// TwinCAT 3 PLC project AlarmsHandler
// Title: AlarmsHandler
// Company: Marden Edwards
// Author: Wiktor Pytka
// ProjectVersion: 1.0.0.0
// ProgramVersion: 3.1.4026.19
// libraries:
//   Tc2_MC2, * (Beckhoff Automation GmbH)
//   Tc2_SerialCom, * (Beckhoff Automation GmbH)
//   Tc2_Standard, * (Beckhoff Automation GmbH)
//   Tc2_System, * (Beckhoff Automation GmbH)
//   Tc2_TcpIp, * (Beckhoff Automation GmbH)
//   Tc2_Utilities, * (Beckhoff Automation GmbH)
// project tree:
//   DUTs/METS/ADS Symobol/ E_SYMBOL_AccessState.TcDUT, E_SYMBOL_AdsStates.TcDUT, ST_SYMBOL_AddressInfo.TcDUT (not stored)
//   DUTs/METS/AI Codes And Validation/ E_CodeAI.TcDUT (not stored), E_CodeType.TcDUT, ST_CodeInfo.TcDUT, ST_CodeValidation.TcDUT (not stored), ST_RejectItems.TcDUT, ST_RejectReasonsForCase.TcDUT (not stored), ST_RejectReasonsForOuter.TcDUT (not stored), ST_RejectReasonsForPack.TcDUT (not stored)
//   DUTs/METS/AI Codes And Validation/GS1_Standard/ E_GS1_CodeAIType.TcDUT (not stored), E_GS1_CodeLvl.TcDUT (not stored), ST_GS1_AI_Attributs.TcDUT (not stored), ST_GS1_AI_Definition.TcDUT (not stored), ST_GS1_CodeInfo.TcDUT (not stored), ST_GS1_CodeValidation.TcDUT (not stored), ST_GS1_Decode_AI.TcDUT (not stored)
//   DUTs/METS/Alarms/ E_MessageID.TcDUT, E_MessageType.TcDUT (not stored), ST_AlarmDB.TcDUT (not stored), ST_Alarms.TcDUT (not stored), ST_AlarmSettings.TcDUT, ST_AlarmsTable.TcDUT (not stored), ST_AlarmStatus.TcDUT (not stored), ST_ALARM_Aux.TcDUT (not stored)
//   DUTs/METS/Aliases/ T_CAC_Filename_1.TcDUT (not stored), T_CASE_Barcode_1.TcDUT (not stored), T_Char_1.TcDUT (not stored), T_CHM_Filename_1.TcDUT (not stored), T_CodeBATCH_1.TcDUT (not stored), T_CodeBRAND_1.TcDUT (not stored), T_CodeCRYPTO_1.TcDUT (not stored), T_CodeGTIN_1.TcDUT (not stored), T_CodeMRP_1.TcDUT (not stored), T_CodePIT_1.TcDUT (not stored), T_CodePO_1.TcDUT (not stored), T_CodePRODUCEDATE_1.TcDUT (not stored), T_CodeRSKU_1.TcDUT (not stored), T_CodeURL_1.TcDUT (not stored), T_DB_LongSTRING_1.TcDUT (not stored), T_FileExtension_1.TcDUT (not stored), T_FolderName_1.TcDUT (not stored), T_FolderPath_1.TcDUT (not stored), T_FSS_RejecCode_1.TcDUT (not stored), T_HMI_PACK_Barcode_1.TcDUT (not stored), T_ISO8601Time_1.TcDUT (not stored), T_LongSTRING_1.TcDUT (not stored), T_OAC_Filename_1.TcDUT (not stored), T_OCV_Filename_1.TcDUT (not stored), T_OHM_Filename_1.TcDUT (not stored), T_OUTER_Barcode_1.TcDUT (not stored), T_PACK_Barcode_1.TcDUT (not stored), T_PCM_Filename_1.TcDUT (not stored), T_PositiveDINT_1.TcDUT (not stored), T_PositiveINT_1.TcDUT (not stored), T_ProductDescription_1.TcDUT (not stored), T_RejectCode_1.TcDUT (not stored), T_TimeLog_1.TcDUT (not stored)
//   DUTs/METS/Case/CAC/ E_CAC_State.TcDUT (not stored), ST_CAC_Data.TcDUT (not stored)
//   DUTs/METS/Case/CHM/CHM Data Structure/GenericHierarchy/Case Item Structures/ ST_CaseContent.TcDUT (not stored), ST_CaseIdentity.TcDUT (not stored), ST_CaseItem.TcDUT (not stored)
//   DUTs/METS/Case/CHM/CHM Data Structure/GenericHierarchy/Outer Item Structures/ ST_OuterContent.TcDUT (not stored), ST_OuterIdentity.TcDUT (not stored), ST_OuterItem.TcDUT (not stored)
//   DUTs/METS/Case/CHM/CHM Data Structure/GenericHierarchy/Pack Item Structures/ ST_PackIdentity.TcDUT (not stored), ST_PackItem.TcDUT (not stored)
//   DUTs/METS/Case/CHM/CHM Data Structure/GenericHierarchy/ ST_DefaultIdentity.TcDUT (not stored)
//   DUTs/METS/Case/CHM/CHM Data Structure/ ST_Attributes.TcDUT (not stored), ST_CHM_GenericHierarchy.TcDUT (not stored) (excluded from build), ST_GenericHierarchy.TcDUT (not stored), ST_MessageHeader.TcDUT (not stored)
//   DUTs/METS/Case/CHM/ E_CHM_GeneratorState.TcDUT (not stored), E_CHM_State.TcDUT (not stored), E_CHM_WriteMode.TcDUT (not stored) (excluded from build), ST_CHM_Data.TcDUT (not stored)
//   DUTs/METS/Case/ E_CASE_State.TcDUT (not stored), ST_CasePackerInfo.TcDUT (not stored), ST_CASE_CaseQueue.TcDUT (not stored), ST_CASE_DefferOuter.TcDUT (not stored), ST_CASE_InfeedQueue.TcDUT (not stored), ST_CASE_OperationData.TcDUT (not stored)
//   DUTs/METS/Case/ORCA/ E_ORCA_State.TcDUT (not stored), ST_ORCA_BrandInfo.TcDUT (not stored), ST_ORCA_Data.TcDUT (not stored), ST_ORCA_Outers.TcDUT (not stored), ST_ORCA_ProductInfo.TcDUT (not stored), ST_ORCA_SiteInfo.TcDUT (not stored)
//   DUTs/METS/Device/CX Unit/Device/ E_CX_DeviceState.TcDUT (not stored)
//   DUTs/METS/Device/CX Unit/EtherCAT/ E_CX_EtherCATState.TcDUT (not stored), ST_CX_EtherCATDeviceState.TcDUT (not stored), ST_CX_EtherCATMasterPNetState.TcDUT (not stored), ST_CX_EtherCATMasterState.TcDUT (not stored)
//   DUTs/METS/Device/CX Unit/EtherCAT/Terminal FBs/EBUS/ ST_EBUS_AnalogueDataIn.TcDUT (not stored), ST_EBUS_EtherCATState.TcDUT (not stored)
//   DUTs/METS/Device/CX Unit/EtherCAT/Terminal FBs/KBUS/ E_KBUS_RegisterAccessState.TcDUT (not stored), ST_KBUS_AnalogueDataIn.TcDUT (not stored), ST_KBUS_AnalogueDataOut.TcDUT (not stored), ST_KBUS_KL1501DataIn.TcDUT (not stored), ST_KBUS_KL1501DataOut.TcDUT (not stored), ST_KBUS_KL5001Config.TcDUT (not stored)
//   DUTs/METS/Device/CX Unit/EtherCAT/Terminal FBs/ ST_EtherCATSlaveInfo.TcDUT (not stored), ST_EtherCATStatus.TcDUT (not stored)
//   DUTs/METS/Device/CX Unit/Network/ E_CX_NetworkInfoState.TcDUT (not stored), E_CX_SetAMSNetIDState.TcDUT (not stored), ST_CX_AdapterInfo.TcDUT (not stored), ST_CX_NetworkInfo.TcDUT (not stored)
//   DUTs/METS/Device/CX Unit/NOVRAM/ E_CX_NVDataCtrlState.TcDUT (not stored), E_CX_NVDataOpMode.TcDUT (not stored), E_CX_NVXMLState.TcDUT (not stored), ST_CX_AMSAddress.TcDUT (not stored), ST_CX_EL6080DataIn.TcDUT (not stored), ST_CX_EL6080DataOut.TcDUT (not stored), ST_CX_NVDataBlock.TcDUT (not stored)
//   DUTs/METS/Device/CX Unit/System/ E_CX_HWType.TcDUT (not stored), E_CX_State.TcDUT (not stored)
//   DUTs/METS/Device/Cylinders/ E_CYLINDER_Name.TcDUT (not stored), E_CYLINDER_Position.TcDUT (not stored), ST_CYLINDER_Config.TcDUT (not stored), ST_CYLINDER_Control.TcDUT (not stored), ST_CYLINDER_IN.TcDUT (not stored), ST_CYLINDER_OUT.TcDUT (not stored), ST_CYLINDER_Status.TcDUT (not stored), ST_CYLINDER_TagID.TcDUT (not stored)
//   DUTs/METS/Device/DB/ E_DB_ScanState.TcDUT (not stored), ST_DB_CACDataCtrl.TcDUT (not stored), ST_DB_OACDataCtrl.TcDUT (not stored), ST_DB_OCVDataCtrl.TcDUT (not stored)
//   DUTs/METS/Device/DB/OLD/ ST_DBResult.TcDUT (not stored) (excluded from build), ST_DB_CACCheckCtrl.TcDUT (not stored) (excluded from build), ST_DB_Config.TcDUT (not stored), ST_DB_OACCheckCtrl.TcDUT (not stored) (excluded from build), ST_DB_OCVCheckCtrl.TcDUT (not stored) (excluded from build), ST_DB_PcvCheckCtrl.TcDUT (not stored) (excluded from build), ST_DB_ReportDBCtrl.TcDUT (not stored), ST_DB_ReportResult.TcDUT (not stored)
//   DUTs/METS/Device/Drive/Analog/Config/ ST_AnalogDrive.TcDUT (not stored)
//   DUTs/METS/Device/Drive/Analog/ ST_DriveCtrl.TcDUT (not stored), ST_PhtcCtrl.TcDUT (not stored) (excluded from build)
//   DUTs/METS/Device/Drive/MC2/Axis Control/ E_AXIS_MotionType.TcDUT (not stored), ST_AXIS_Control.TcDUT (not stored), ST_AXIS_IN.TcDUT (not stored), ST_AXIS_OUT.TcDUT (not stored), ST_AXIS_Status.TcDUT (not stored)
//   DUTs/METS/Device/Drive/MC2/Config/ ST_AXIS_Config.TcDUT (not stored)
//   DUTs/METS/Device/Drive/MC2/EtherCAT/AX5000 FBs/ ST_AX5000_TouchProbe.TcDUT (not stored)
//   DUTs/METS/Device/Drive/MC2/EtherCAT/Encoder FBs/ ST_DeviceAddress.TcDUT (not stored)
//   DUTs/METS/Device/Drive/MC2/ E_MC_Name.TcDUT (not stored)
//   DUTs/METS/Device/Drive/MC2/NC Axis/Cam/ E_CAM_Update.TcDUT (not stored)
//   DUTs/METS/Device/Drive/MC2/NC Axis/ E_AXIS_CtrlState.TcDUT (not stored), E_TORQUE_Scaling.TcDUT (not stored), ST_AxisCtrlRamps.TcDUT (not stored), ST_DriveStatus.TcDUT (not stored), ST_LatchPosBuffer.TcDUT (not stored), ST_NC_EncDataIn.TcDUT (not stored), ST_NC_EncDataOut.TcDUT (not stored)
//   DUTs/METS/Device/Drive/MC2/TempAxis/ ST_AxisHomeStruct.TcDUT (not stored) (excluded from build), ST_AxisMotionStruct.TcDUT (not stored) (excluded from build)
//   DUTs/METS/Device/Drive/Profinet/Config/ ST_ProfinetDrive.TcDUT (not stored), ST_ProfinetMasterConfig.TcDUT (not stored)
//   DUTs/METS/Device/Drive/Profinet/ E_DRIVE_Name.TcDUT (not stored), ST_PNetMasterStatus.TcDUT (not stored)
//   DUTs/METS/Device/Drive/Profinet/Parameters/ ST_DataPntAdr.TcDUT (not stored), ST_KeyPadDisplay.TcDUT (not stored), ST_Parameter.TcDUT (not stored), ST_ParameterControl.TcDUT (not stored), ST_Parameters.TcDUT (not stored), ST_Value.TcDUT (not stored)
//   DUTs/METS/Device/Drive/Profinet/_G120/Drives/ E_DRIVE_DataType.TcDUT (not stored), ST_DRIVE_INPUT.TcDUT (not stored), ST_DRIVE_OUTPUT.TcDUT (not stored), ST_DRIVE_STATUS.TcDUT (not stored), ST_G120_ExtendedIn.TcDUT (not stored), ST_G120_ExtendedOut.TcDUT (not stored), ST_G120_IN.TcDUT (not stored), ST_G120_OUT.TcDUT (not stored), ST_G120_Status.TcDUT (not stored)
//   DUTs/METS/Device/Drive/Profinet/_G120/ ST_G120_Control.TcDUT (not stored)
//   DUTs/METS/Device/Encoders/CAMS/ ST_AFS60_Cam.TcDUT (not stored), ST_AFS60_CamHMi.TcDUT (not stored), ST_AFS60_Config.TcDUT (not stored), ST_AFS60_Status.TcDUT (not stored)
//   DUTs/METS/Device/Encoders/ E_ENOCDER_Name.TcDUT (not stored), ST_ENCODER_IN.TcDUT (not stored), ST_ENCODER_OUT.TcDUT (not stored), ST_ENCODER_Status.TcDUT (not stored)
//   DUTs/METS/Device/IO2 Controls/ E_IO2_InputSource.TcDUT (not stored), E_IO2_Type.TcDUT (not stored), ST_IO2_Diagnostic.TcDUT (not stored), ST_IO2_InputPLC.TcDUT (not stored), ST_IO2_OutputPLC.TcDUT (not stored)
//   DUTs/METS/Device/IO2 Controls/Input Ctrl/ ST_IO2_DoubleInputCtrl.TcDUT (not stored), ST_IO2_DoubleInputLockedCtrl.TcDUT (not stored), ST_IO2_SingleInputCtrl.TcDUT (not stored), ST_IO2_SingleInputLockedCtrl.TcDUT (not stored)
//   DUTs/METS/Device/IO2 Controls/Outpout Ctrl/ ST_IO2_OutputCtrl.TcDUT (not stored)
//   DUTs/METS/Device/Printers/ E_PRINTER_Name.TcDUT (not stored), E_PRINTER_State.TcDUT (not stored), ST_PRINTER_Config.TcDUT (not stored), ST_PRINTER_IN.TcDUT (not stored), ST_PRINTER_OUT.TcDUT (not stored), ST_PRINTER_Status.TcDUT (not stored)
//   DUTs/METS/Device/Scanner/ E_ClientSteps.TcDUT (not stored), E_DataExchaSteps.TcDUT (not stored), E_SCANNER_CodeType.TcDUT (not stored), E_SCANNER_DeviceType.TcDUT (not stored), E_SCANNER_Name.TcDUT (not stored), E_SCANNER_State.TcDUT (not stored), E_SCANNER_Vendor.TcDUT (not stored), ST_SCANNER.TcDUT (not stored), ST_SCANNER_ApplicationIdentifier.TcDUT (not stored), ST_SCANNER_CameraMap.TcDUT (not stored), ST_SCANNER_CodeData.TcDUT (not stored), ST_SCANNER_Config.TcDUT (not stored), ST_SCANNER_Evaluation.TcDUT (not stored), ST_SCANNER_ImageData.TcDUT (not stored), ST_SCANNER_ManualCtrl.TcDUT (not stored), ST_SCANNER_OpState.TcDUT (not stored), ST_SCANNER_Options.TcDUT (not stored), ST_SCANNER_Performance.TcDUT (not stored), ST_SCANNER_Statistics.TcDUT (not stored), ST_SCANNER_TriggerID.TcDUT (not stored)
//   DUTs/METS/Device/Scanner/Hand Scanner/ E_ConnectSteps.TcDUT (not stored), E_DataSequence.TcDUT (not stored), E_SCANNER_Baudrate.TcDUT (not stored), ST_SCANNER_HoneywellConfig.TcDUT (not stored), ST_SCANNER_HoneywellCtrl.TcDUT (not stored), ST_SCANNER_HoneywellStatus.TcDUT (not stored), ST_SCANNER_HostAck.TcDUT (not stored), ST_SCANNER_USBConfig.TcDUT (not stored)
//   DUTs/METS/Device/Scanner/NewModel/ ST_SCANNER_Configuration.TcDUT, ST_SCANNER_Ctrl.TcDUT (not stored), ST_SCANNER_CtrlMapping.TcDUT (not stored), ST_SCANNER_CtrlOptions.TcDUT (not stored) (excluded from build), ST_SCANNER_IN.TcDUT (not stored), ST_SCANNER_ManualStatus.TcDUT (not stored), ST_SCANNER_OUT.TcDUT (not stored), ST_SCANNER_Status.TcDUT (not stored)
//   DUTs/METS/Files/ E_FILE_CtrlState.TcDUT (not stored), E_FILE_DeleteOldFilesState.TcDUT (not stored), E_FILE_State.TcDUT (not stored), ST_FILE_WriteFileStatistic.TcDUT (not stored)
//   DUTs/METS/HMI/Device Manual Control/ ST_HMI_AxisCtrl.TcDUT (not stored), ST_HMI_CylinderCtrl.TcDUT (not stored), ST_HMI_G120Ctrl.TcDUT (not stored), ST_HMI_PrinterCtrl.TcDUT (not stored)
//   DUTs/METS/HMI/Device Status/ E_HMI_DriveStatus.TcDUT, ST_HMI_AxisStatus.TcDUT (not stored), ST_HMI_CylinderStatus.TcDUT (not stored), ST_HMI_G120Status.TcDUT (not stored), ST_HMI_HoneywellStatus.TcDUT (not stored), ST_HMI_PrinterStatus.TcDUT (not stored)
//   DUTs/METS/HMI/HMIQueue/ ST_HMI_CAC_Data.TcDUT (not stored), ST_HMI_CaseRejectCode.TcDUT (not stored), ST_HMI_CaseVerifiedCode.TcDUT (not stored), ST_HMI_CASE_CaseQueue.TcDUT (not stored), ST_HMI_InfeedQueue.TcDUT (not stored), ST_HMI_OAC_Data.TcDUT (not stored), ST_HMI_OCV_Data.TcDUT (not stored), ST_HMI_OuterStatus.TcDUT (not stored), ST_HMI_PACK_BufferStatus.TcDUT (not stored), ST_HMI_PLAS_Queue.TcDUT (not stored)
//   DUTs/METS/HMI/ ST_HMI_BarGraph.TcDUT (not stored), ST_HMI_Buttons.TcDUT (not stored), ST_HMI_CSVStoreTable.TcDUT (not stored), ST_HMI_StationStatus.TcDUT (not stored), ST_HMI_Visualisation.TcDUT (not stored)
//   DUTs/METS/KPI/ ST_KPI_CasePackerSignals.TcDUT (not stored), ST_KPI_CodePos.TcDUT (not stored), ST_KPI_InspectionEfficency.TcDUT (not stored), ST_KPI_ItemsProduced.TcDUT (not stored), ST_KPI_OCVFile.TcDUT (not stored), ST_KPI_OutersProcessing.TcDUT (not stored), ST_KPI_OutersProduced.TcDUT (not stored)
//   DUTs/METS/LogData/ E_LOG_Handler.TcDUT (not stored), ST_LOG_Alarms.TcDUT (not stored), ST_LOG_EventData.TcDUT (not stored), ST_LOG_FileWriteError.TcDUT (not stored), ST_LOG_MachineState.TcDUT (not stored), ST_LOG_RejectReasons.TcDUT (not stored), ST_LOG_WriteImageData.TcDUT (not stored)
//   DUTs/METS/NV Data/ ST_NOVRAM_METS_Cameras.TcDUT (not stored), ST_NOVRAM_METS_CaseInspactionLog.TcDUT (not stored), ST_NOVRAM_METS_DualInputs.TcDUT (not stored), ST_NOVRAM_METS_EventCounters.TcDUT (not stored), ST_NOVRAM_METS_Inspection.TcDUT (not stored)
//   DUTs/METS/Outers/ E_OUTER_AgrregationState.TcDUT (not stored), E_OUTER_State.TcDUT (not stored), ST_OUTER_Status.TcDUT (not stored)
//   DUTs/METS/Outers/OAC/ E_OAC_State.TcDUT (not stored), ST_OAC_Data.TcDUT (not stored)
//   DUTs/METS/Outers/SFLX/ E_SIDEFLEX_UnitType.TcDUT (not stored), ST_SIDEFLEX_Offset.TcDUT (not stored), ST_SIDEFLEX_ProcessData.TcDUT (not stored)
//   DUTs/METS/Packs/ E_OCV_CheckMode.TcDUT (not stored), E_OCV_State.TcDUT (not stored), E_PACK_FilledInStatus.TcDUT (not stored), E_PACK_ReadStep.TcDUT (not stored), E_PACK_State.TcDUT (not stored), ST_PACK_CodeBuffer.TcDUT (not stored), ST_PACK_CodeStatus.TcDUT (not stored), ST_PACK_ConfirmationQueue.TcDUT (not stored), ST_PACK_Data.TcDUT (not stored), ST_PACK_DuplicatesCheck.TcDUT (not stored), ST_PACK_InfeedQueue.TcDUT (not stored), ST_PACK_InTransferQueue.TcDUT (not stored), ST_PACK_LastFilledCodes.TcDUT (not stored), ST_PACK_TriggerOffset.TcDUT (not stored)
//   DUTs/METS/Packs/_Lab/ ST_LAB_OuterData.TcDUT (not stored), ST_LAB_PackData.TcDUT (not stored)
//   DUTs/METS/PCM/ E_PCM_State.TcDUT (not stored), ST_PCM_Data.TcDUT (not stored), ST_PCM_Status.TcDUT (not stored)
//   DUTs/METS/PCM/PCM_Hierarchy/ProductInformation/Product/ ST_HierarchyData.TcDUT (not stored), ST_HierarchyDataList.TcDUT (not stored)
//   DUTs/METS/PCM/PCM_Hierarchy/ProductInformation/Settings/ ST_ToleranceThresholdCS.TcDUT (not stored), ST_ToleranceThresholdOUT.TcDUT (not stored), ST_ToleranceThresholdPK.TcDUT (not stored)
//   DUTs/METS/PCM/PCM_Hierarchy/ProductInformation/ ST_PCMProduct.TcDUT (not stored), ST_PCMSettings.TcDUT (not stored)
//   DUTs/METS/PCM/PCM_Hierarchy/ ST_PCMMessageHeader.TcDUT (not stored), ST_ProductInformation.TcDUT (not stored)
//   DUTs/METS/String Processing/ E_STRING_ExtrMode.TcDUT (not stored)
//   DUTs/METS/System/ E_SYSTEM_CTState.TcDUT (not stored), E_SYSTEM_HandScannerBaudrate.TcDUT (not stored), E_SYSTEM_ItemType.TcDUT (not stored), E_SYSTEM_MachineState.TcDUT (not stored), E_SYSTEM_MaintainFolders.TcDUT (not stored), E_SYSTEM_OSType.TcDUT (not stored), ST_SYSTEM_Config.TcDUT, ST_SYSTEM_DateTime.TcDUT (not stored), ST_SYSTEM_DeviceState.TcDUT (not stored), ST_SYSTEM_Door.TcDUT (not stored), ST_SYSTEM_MachineID.TcDUT (not stored), ST_SYSTEM_MachineMode.TcDUT (not stored), ST_SYSTEM_MachineState.TcDUT (not stored), ST_SYSTEM_ProductionLine.TcDUT (not stored), ST_SYSTEM_SafetyStatus.TcDUT (not stored), ST_SYSTEM_SoftwareVersion.TcDUT (not stored)
//   DUTs/METS/System/Status/ ST_SYSTEM_ArchiveDBStatus.TcDUT (not stored), ST_SYSTEM_BridgeStatus.TcDUT (not stored), ST_SYSTEM_LoggerStatus.TcDUT (not stored), ST_SYSTEM_MachineStatus.TcDUT (not stored), ST_SYSTEM_ReportingDBStatus.TcDUT (not stored)
//   DUTs/METS/System/System Modes/ E_SYSTEM_AutomationMode.TcDUT (not stored), E_SYSTEM_OuterAggregationMode.TcDUT (not stored), E_SYSTEM_PackAggregationMode.TcDUT (not stored)
//   DUTs/METS/TCPIP Address/ E_TCPIP_State.TcDUT, ST_TCPIP_AddressPort.TcDUT (not stored)
//   DUTs/METS/XML Processing/ E_XML_CtrlState.TcDUT (not stored), E_XML_GeneratorState.TcDUT (not stored), E_XML_WritingMode.TcDUT (not stored)
//   DUTs/METS/_StationOperational/C715 Tempalate Example/ E_04_ElevatorState_C715.TcDUT (not stored), E_Axis_C715.TcDUT (not stored), E_Cylinder_C715.TcDUT (not stored), ST_04_ElevatorSeq_C715.TcDUT (not stored), ST_BundleTrackingRegister_C715.TcDUT (not stored), ST_CommonStationConfig_C715.TcDUT (not stored)
//   DUTs/METS/_StationOperational/ E_00_StationStateTemplate.TcDUT (not stored), ST_00_StationStructTemplate.TcDUT (not stored)
//   DUTs/METS/_StationOperational/Manual Machine/ E_OuterPrintStationState.TcDUT (not stored), ST_OuterPrintStationStruct.TcDUT (not stored)
//   DUTs/METS/_StationOperational/SeqCtrl/ ST_STATION_Requests.TcDUT (not stored), ST_STATION_Status.TcDUT (not stored)
//   GVLs/Global Variables/Aliases/ T_CAC_Filename.TcDUT, T_CASE_Barcode.TcDUT, T_Char.TcDUT, T_CHM_Filename.TcDUT, T_CodeBATCH.TcDUT, T_CodeBRAND.TcDUT, T_CodeCRYPTO.TcDUT, T_CodeGTIN.TcDUT, T_CodeMRP.TcDUT, T_CodePIT.TcDUT, T_CodePO.TcDUT, T_CodePRODUCEDATE.TcDUT, T_CodeRSKU.TcDUT, T_CodeURL.TcDUT, T_DB_LongSTRING.TcDUT, T_FileExtension.TcDUT, T_FolderName.TcDUT, T_FolderPath.TcDUT, T_FSS_RejecCode.TcDUT, T_HMI_PACK_Barcode.TcDUT, T_ISO8601Time.TcDUT, T_LongSTRING.TcDUT, T_OAC_Filename.TcDUT, T_OCV_Filename.TcDUT, T_OHM_Filename.TcDUT, T_OUTER_Barcode.TcDUT, T_PACK_Barcode.TcDUT, T_PCM_Filename.TcDUT, T_PositiveDINT.TcDUT, T_PositiveINT.TcDUT, T_ProductDescription.TcDUT, T_RejectCode.TcDUT, T_TimeLog.TcDUT
//   GVLs/Global Variables/ gConstants.TcGVL (not stored), gHMI.TcGVL (not stored), gIOFiltered.TcGVL (not stored), gMessage.TcGVL, gNovRAM.TcGVL (not stored), gPersistent.TcGVL (not stored)
//   GVLs/Global Variables/InputsOutputsDT/ gCamDevice.TcGVL (not stored), IOVarDT_H.TcGVL (not stored), IOVarDT_S.TcGVL (not stored), _Labs.TcGVL (not stored)
//   GVLs/Global Variables/InputsOutputs_CML/ IOVariablesCX_CML.TcGVL (excluded from build), IOVariablesEUCA_CML.TcGVL (excluded from build), IOVariablesPACAN_CML.TcGVL (excluded from build), IOVariablesPAOL_CML.TcGVL (excluded from build), IOVariablesPLAS_CML.TcGVL (excluded from build)
//   GVLs/Global Variables/InputsOutputs_OC/ IOVariablesCX_OC.TcGVL (excluded from build), IOVariablesEUCA_OC.TcGVL (excluded from build), IOVariablesPAOL_OC.TcGVL (excluded from build), IOVariablesPLAS_OC.TcGVL (excluded from build)
//   GVLs/Global Variables/InputsOutputs_SFLX/ IOVariablesCX_SFLX.TcGVL (excluded from build), IOVariablesEUCA_SFLX.TcGVL (excluded from build), IOVariablesPAOL_SFLX.TcGVL (excluded from build), IOVariablesPLAS_SFLX.TcGVL (excluded from build)
//   GVLs/Global Variables/METS/ gDevice.TcGVL (not stored), gProcess.TcGVL (not stored)
//   GVLs/Global Variables/_VERSION/ _VERSION_CONTROL.TcGVL
//   POUs/Alarm/ FB_ALARM_GroupManagment.TcPOU (not stored), FB_ALARM_Handler.TcPOU (not stored), FB_ALARM_LogTable.TcPOU (not stored), F_ALARM_SetDefinition.TcPOU
//   POUs/Utilities/Concat Function/ F_CONCAT3.TcPOU (not stored), F_CONCAT4.TcPOU (not stored), F_CONCAT5.TcPOU (not stored), F_CONCAT6.TcPOU (not stored), F_CONCAT7.TcPOU (not stored), F_CONCAT8.TcPOU (not stored), F_CONCAT9.TcPOU (not stored)
//   Version/ Global_Version.TcGVL
// real-time tasks:
//   TASK TcUnit_Task: cycle T#10ms, priority 10, ADS port 350

// ---- DUTs/METS/ADS Symobol/E_SYMBOL_AccessState.TcDUT
{attribute 'qualified_only'}
TYPE E_SYMBOL_AccessState :
(
	E_SYMBOL_IDLE,
	E_SYMBOL_GETSYMBOLINFO,
	E_SYMBOL_READDATA,
	E_SYMBOL_WRITEDATA,
	E_SYMBOL_DONE
);
END_TYPE

// ---- DUTs/METS/ADS Symobol/E_SYMBOL_AdsStates.TcDUT
{attribute 'qualified_only'}
TYPE E_SYMBOL_AdsStates :
(
	ADSSTATES_INVALID :=0,
	ADSSTATES_IDLE :=1,
	ADSSTATES_RESET :=2,
	ADSSTATES_INIT :=3,
	ADSSTATES_START :=4,
	ADSSTATES_RUN :=5,
	ADSSTATES_STOP :=6,
	ADSSTATES_SAVECFG :=7,
	ADSSTATES_LOADCFG :=8,
	ADSSTATES_POWERFAILURE :=9,
	ADSSTATES_POWERGOOD :=10,
	ADSSTATES_ERROR :=11
);
END_TYPE

// ---- DUTs/METS/AI Codes And Validation/E_CodeType.TcDUT
{attribute 'qualified_only'}
TYPE E_CodeType :
(
	E_NONE,
	E_PACK,
	E_INTERIM,
	E_OUTER,
	E_CASE
);
END_TYPE

// ---- DUTs/METS/AI Codes And Validation/ST_CodeInfo.TcDUT
TYPE ST_CodeInfo :
STRUCT
	eCodeType					:	E_CodeType;

	nMinLength					: 	INT;
	nEntireLength				:	INT;
	bValidateEntireLength		: 	BOOL;
	nNumberOfAIs				:	INT;

	stGTIN 						:	ST_CodeValidation	:=		(sFieldName :='GTIN',				bNameEditable := FALSE, 	nGS1_AI := 1);
	stBatchID 					:	ST_CodeValidation	:=		(sFieldName :='BatchID', 			bNameEditable := FALSE, 	nGS1_AI := 10);
	stSerialCode 				:	ST_CodeValidation	:=		(sFieldName :='SerialCode', 		bNameEditable := FALSE, 	nGS1_AI := 21);
	stProductionOrder 			:	ST_CodeValidation	:=		(sFieldName :='ProductionOrder', 	bNameEditable := FALSE, 	nGS1_AI := 91);
	stCryptoCode				:	ST_CodeValidation	:=		(sFieldName :='CryptoCode', 		bNameEditable := FALSE, 	nGS1_AI := 93);
	stRSKU						:	ST_CodeValidation	:=		(sFieldName :='RSKU', 				bNameEditable := FALSE, 	nGS1_AI := 240);
	stMRP		 				:	ST_CodeValidation	:=		(sFieldName :='MRP', 				bNameEditable := FALSE, 	nGS1_AI := 8005);
	stBrandSpecification		:	ST_CodeValidation	:=		(sFieldName :='BrandSpec',			bNameEditable := FALSE, 	nGS1_AI := 92);
	stProduceDate				:	ST_CodeValidation	:=		(sFieldName :='ProduceDate',		bNameEditable := TRUE, 		nGS1_AI := 94);
	stUserField					:	ST_CodeValidation	:=		(sFieldName :='',					bNameEditable := TRUE, 		nGS1_AI := 95);

END_STRUCT
END_TYPE

// ---- DUTs/METS/AI Codes And Validation/ST_RejectItems.TcDUT
TYPE ST_RejectItems :
STRUCT
	nRejectID			: UINT;
	sMetsDisplayCode	: T_RejectCode; (*this is what is displayed on our HMI - nn is replaced by the number of failures/successes*)
	sMetsSearchCode	: STRING(50); (*this is what to search for when changing the reject reason for FSS*)
	sFssSendCode		: T_FSS_RejecCode; (*this is what to send to FSS*)
END_STRUCT
END_TYPE

// ---- DUTs/METS/Alarms/E_MessageID.TcDUT
{attribute 'qualified_only'}
{attribute 'to_string'}
TYPE E_MessageID :
(
	MSG_000 := 0,
	MSG_001,
	MSG_002,
	MSG_003,
	MSG_004,
	MSG_005,
	MSG_006,
	MSG_007,
	MSG_008,
	MSG_009,
	MSG_010,
	MSG_011,
	MSG_012,
	MSG_013,
	MSG_014,
	MSG_015,
	MSG_016,
	MSG_017,
	MSG_018,
	MSG_019,
	MSG_020,
	MSG_021,
	MSG_022,
	MSG_023,
	MSG_024,
	MSG_025,
	MSG_026,
	MSG_027,
	MSG_028,
	MSG_029,
	MSG_030,
	MSG_031,
	MSG_032,
	MSG_033,
	MSG_034,
	MSG_035,
	MSG_036,
	MSG_037,
	MSG_038,
	MSG_039,
	MSG_040,
	MSG_041,
	MSG_042,
	MSG_043,
	MSG_044,
	MSG_045,
	MSG_046,
	MSG_047,
	MSG_048,
	MSG_049,
	MSG_050,
	MSG_051,
	MSG_052,
	MSG_053,
	MSG_054,
	MSG_055,
	MSG_056,
	MSG_057,
	MSG_058,
	MSG_059,
	MSG_060,
	MSG_061,
	MSG_062,
	MSG_063,
	MSG_064,
	MSG_065,
	MSG_066,
	MSG_067,
	MSG_068,
	MSG_069,
	MSG_070,
	MSG_071,
	MSG_072,
	MSG_073,
	MSG_074,
	MSG_075,
	MSG_076,
	MSG_077,
	MSG_078,
	MSG_079,
	MSG_080,
	MSG_081,
	MSG_082,
	MSG_083,
	MSG_084,
	MSG_085,
	MSG_086,
	MSG_087,
	MSG_088,
	MSG_089,
	MSG_090,
	MSG_091,
	MSG_092,
	MSG_093,
	MSG_094,
	MSG_095,
	MSG_096,
	MSG_097,
	MSG_098,
	MSG_099,
	MSG_100,
	MSG_101,
	MSG_102,
	MSG_103,
	MSG_104,
	MSG_105,
	MSG_106,
	MSG_107,
	MSG_108,
	MSG_109,
	MSG_110,
	MSG_111,
	MSG_112,
	MSG_113,
	MSG_114,
	MSG_115,
	MSG_116,
	MSG_117,
	MSG_118,
	MSG_119,
	MSG_120,
	MSG_121,
	MSG_122,
	MSG_123,
	MSG_124,
	MSG_125,
	MSG_126,
	MSG_127,
	MSG_128,
	MSG_129,
	MSG_130,
	MSG_131,
	MSG_132,
	MSG_133,
	MSG_134,
	MSG_135,
	MSG_136,
	MSG_137,
	MSG_138,
	MSG_139,
	MSG_140,
	MSG_141,
	MSG_142,
	MSG_143,
	MSG_144,
	MSG_145,
	MSG_146,
	MSG_147,
	MSG_148,
	MSG_149,
	MSG_150,
	MSG_151,
	MSG_152,
	MSG_153,
	MSG_154,
	MSG_155,
	MSG_156,
	MSG_157,
	MSG_158,
	MSG_159,
	MSG_160,
	MSG_161,
	MSG_162,
	MSG_163,
	MSG_164,
	MSG_165,
	MSG_166,
	MSG_167,
	MSG_168,
	MSG_169,
	MSG_170,
	MSG_171,
	MSG_172,
	MSG_173,
	MSG_174,
	MSG_175,
	MSG_176,
	MSG_177,
	MSG_178,
	MSG_179,
	MSG_180,
	MSG_181,
	MSG_182,
	MSG_183,
	MSG_184,
	MSG_185,
	MSG_186,
	MSG_187,
	MSG_188,
	MSG_189,
	MSG_190,
	MSG_191,
	MSG_192,
	MSG_193,
	MSG_194,
	MSG_195,
	MSG_196,
	MSG_197,
	MSG_198,
	MSG_199,
	MSG_200,
	MSG_201,
	MSG_202,
	MSG_203,
	MSG_204,
	MSG_205,
	MSG_206,
	MSG_207,
	MSG_208,
	MSG_209,
	MSG_210,
	MSG_211,
	MSG_212,
	MSG_213,
	MSG_214,
	MSG_215,
	MSG_216,
	MSG_217,
	MSG_218,
	MSG_219,
	MSG_220,
	MSG_221,
	MSG_222,
	MSG_223,
	MSG_224,
	MSG_225,
	MSG_226,
	MSG_227,
	MSG_228,
	MSG_229,
	MSG_230,
	MSG_231,
	MSG_232,
	MSG_233,
	MSG_234,
	MSG_235,
	MSG_236,
	MSG_237,
	MSG_238,
	MSG_239,
	MSG_240,
	MSG_241,
	MSG_242,
	MSG_243,
	MSG_244,
	MSG_245,
	MSG_246,
	MSG_247,
	MSG_248,
	MSG_249,
	MSG_250,
	MSG_251,
	MSG_252,
	MSG_253,
	MSG_254,
	MSG_255
	
);
END_TYPE

// ---- DUTs/METS/Alarms/ST_AlarmSettings.TcDUT
TYPE ST_AlarmSettings :
STRUCT
	aTextMessageTable		: ARRAY [0..31] OF STRING(200);
	aAlarmTriggerTable		: ARRAY [0..31] OF BOOL;

	aAlarmTimoutTable		: ARRAY [0..31] OF TIME;
	aBlockEnableTable		: ARRAY [0..31] OF BOOL :=[ 32 (FALSE)];
	aInhibitResetTable		: ARRAY [0..31] OF BOOL;
	aAutoResetTable			: ARRAY[0..31] OF BOOL;
	//aInternalResetTable		: ARRAY [0..31] OF BOOL;

	aCategoryNoTable		: ARRAY[0..31] OF INT;
	aMessageTypeStatusTable	: ARRAY[0..31] OF WORD;
END_STRUCT
END_TYPE

// ---- DUTs/METS/Device/Scanner/NewModel/ST_SCANNER_Configuration.TcDUT
TYPE ST_SCANNER_Configuration :     //ST_SCANNER_Config
STRUCT
	sDeviceName				: STRING(30) := 'Camera';
	bDisableCameraUse		: BOOL;
	aCameraWarningLevel		: INT := 90;
	stCameraIP				: ST_TCPIP_AddressPort;
	tTimeOut				: TIME := T#3S;
	eCameraVendor			: E_SCANNER_Vendor;
	sFC1ReplacmentChar		: T_Char;
	bDontParseAsGS1			: BOOL;

	eScannerType			: E_SCANNER_DeviceType;
	eExpectedType			: E_SCANNER_CodeType;
	bUseExternalLight		: BOOL;
	nLightingIntensity		: INT;
	nDisplayDelayConfig		: BOOL;

	nImageBuffer			: INT := 1;
	nExpectedResp			: INT := 1;
END_STRUCT
END_TYPE

// ---- DUTs/METS/HMI/Device Status/E_HMI_DriveStatus.TcDUT
{attribute 'qualified_only'}
TYPE E_HMI_DriveStatus :
(
	UNKNOWN := 0,
	STOPPED := 1,
	RUNNING := 2,
	ERROR 	:= 3
);
END_TYPE

// ---- DUTs/METS/System/ST_SYSTEM_Config.TcDUT
{attribute 'pack_mode' := '1'}
TYPE ST_SYSTEM_Config :
STRUCT
(*******************************************************************************************************************************************************)
(*********************************************************General EUCA-TPD*******************************************************************************)
(*******************************************************************************************************************************************************)
(*General screen*)
	sBackupName								: STRING;
	sProductionSite 							: STRING(4);
	stProductionLine 							: ST_SYSTEM_ProductionLine;
	sShiftOffsetTime							: STRING(6);	(* shift offset time, formatted as '-06:00' or '+02:00' *)
	stSoftVersion								: ST_SYSTEM_SoftwareVersion;

	sFC1ReplacmentChar						: STRING(1) := '';

(*FSS settings*)
	tFSSLostConnectionTimeOut				: TIME := t#30m;
	sFSS_Server_IPAddress						: STRING:= '127.0.0.1'; (*Do not remove. Used for HMI*)
	sFSS_Server_WebRequest					: T_MaxString := 'http://127.0.0.1/Apriso/MessageProcessor/FlexNetMessageProcessor.asmx'; (*Do not removed. Used for HMI - this is the CHM sending endpoint*)
	nFSSResponseTimeout						: UINT := 60000; (*: TIME := t#60s;*)
	nFSSResendAttempts						: INT := 5;

(*Shift Setup schedule*)
	aShiftSchedule								: ARRAY[1..cSHIFTNUMBER] OF TIMESTRUCT;
	aShiftChangeActive							: ARRAY[1..cSHIFTNUMBER] OF BOOL;

(*Door*)
	stDoorSettingsZone1					: ST_SYSTEM_Door;
	stDoorSettingsZone2					: ST_SYSTEM_Door;

(*Barcode setup - NEW - Gradually implementing*)
	stCodeInfo_Pack								: ST_CodeInfo :=		(eCodeType :=E_CodeType.E_PACK);
	stCodeInfo_Intermediate						: ST_CodeInfo :=		(eCodeType :=E_CodeType.E_INTERIM);
	stCodeInfo_Outer								: ST_CodeInfo :=		(eCodeType :=E_CodeType.E_OUTER);
	stCodeInfo_Case								: ST_CodeInfo :=		(eCodeType :=E_CodeType.E_CASE);

(*******************************************************************************************************************************************************)
(********************************************************Switch******************************************************************************)
(*******************************************************************************************************************************************************)
(*General Switches*)
	bEUCAMonitor24VSupply					: BOOL := TRUE;
	bMonitorRemote24VSupply				: BOOL;
	bInhibitSafetyResetWhenAirNOK			: BOOL;

	bKPIRemoteShareEnable					: BOOL;
	bSystemLogEnable							: BOOL := TRUE;
	bArchiveDBEnable							: BOOL := TRUE;
	bPassthrough								: BOOL;
	bPassthroughTPD							: BOOL;
	bHandScannerInMainCabinet				: BOOL; (**)
	bValidateOCVOnly							: BOOL;
	bEnableRestoreOCV						: BOOL;		(*Enable Restoring of OCV data from structure*)
	bATTPModeEnable							: BOOL := TRUE;

	bConditionalStateAllowed					: BOOL := TRUE;
	bNoStationsAvailable						: BOOL := TRUE;
	bCommisioningMode						: BOOL; 	(**)
	bConveyorAsPreMachine					: BOOL := TRUE;

	bExistPreTPDBuildBackSensor				: BOOL := TRUE;
	bExistTPDExitBlockedSensor				: BOOL := TRUE;
	bExistPreEUCABuildBackSensor			: BOOL;
	bExistEUCAExitBlockedSensor				: BOOL;
	bExistWrapperPackRejectSesnor			: BOOL;

(*Enable Master List Fillin*)
	bEnablePackPrimaryMasterList					: BOOL:=TRUE;
	bEnablePackSecondaryMasterList				: BOOL:=TRUE;
	bEnableOuterMasterList						: BOOL:=TRUE;

	bExtendedDiagnosticEnable				: BOOL;
	bDotCodeFormat								: BOOL;
	bQRCodeFormat								: BOOL;

(*Pack*)
	bEnableFastArming							: BOOL:=TRUE;		(*Enable arming sensors even if outer did not leave Lightox yet *)
	bPAOLIsolatorExist						: BOOL;
	bLightbox4TrigerSystemExist				: BOOL;
	bLightboxLensAirExist						: BOOL;
	bLighboxOverCMLConveyor					: BOOL;
	bLightboxCamerasOnFullResolution				: BOOL;
	bCloseCameraRelay						: BOOL;
	bPackSeparatorAnalogControl				: BOOL;
	bCameraOnLeftSide							: BOOL; 	(*Set to true if the camera is on the left hand side of the conveyor as the packs travel trhough it towards the CML*)
	bPackCodesTrailing							: BOOL := TRUE; 	(*Set to true if the pack codes are on the trailing edge of the pack as it travels through the infeed cameras*)
	bFirstPackCodeOnTop							: BOOL;			(*Used for correct mapping packs from pack confirmation camera*)

	bEnableCodeAdjustment						: BOOL;
	bEnableCodeDuplicateCheck					: BOOL;
	bExtendedOCVDupCheck						: BOOL;
	bLinearPackBufferExist							: BOOL;
	bEnableStopForInvalideCode					: BOOL;	(*Stop METS immidiatly after Lightbox detect invalide code*)
	bEnablePackCodeDateCheck					: BOOL;
	bFixedTriggerOffsetEnable						: BOOL;

(*Outer*)
	bFrontConfirmationCameraInUse			: BOOL;				(*Rear confirmation camera 192.168.1.41 = false, front confiramtion camera 192.168.1.42 = true*)
	bEnableOuterRejectConfirmation			: BOOL;
	bEnableOuterTransferConfirmation		: BOOL;
	bMasterListCameraDoubleRead				: BOOL := TRUE;
	bAggregationCameraRunWithTrigger			: BOOL;
	bAggregationStopOnInvalidCode				: BOOL ;
	bUseAuxRowCompleteSesnor					: BOOL;
	bUseInterimCodeForLastPosition				: BOOL;
	bSkipStopGate									: BOOL;
	bPreLabelerShiftRegUsed						: BOOL;
	bConfirmOnOuter								: BOOL;		(*At Focke NCW outer is confirmet by it last packs*)
	bEanbleRestoreOCVFromConfirmation			: BOOL;		(*At Focke NCW two outers will be resotred after index = 2 x pack per outers*)
	bExtendedOACDupCheck						: BOOL;

(*Case*)
	bPushIntoCaseCount							: BOOL;
	bIntermediateBufferExist						: BOOL;
	bCasePackerDirectCutOut						: BOOL;
	bCasePositionOverwritingCheck				: BOOL := TRUE;
	//bAddOACFromFileOnly						: BOOL;	(*Add OAC to infeed from file not from arrOuterStatus*)
	bSentOnlyGoodHierarchy						: BOOL := TRUE;
	bArchiveRejectedHierarchy					: BOOL := TRUE;
	bEnableStopOnOverWrittenData				: BOOL;
	bResetPushCountOnDoorOpen				: BOOL;
	bCheckDuplicateCaseLabel					: BOOL;
	bManualConfirmationEnable					: BOOL;
	bEnableStopOnCaseInavlid						: BOOL;
	bUseCaseFullAsValidationTrigger				: BOOL;
	bUseCaseContentReject						: BOOL;
	bUseRejectByCasepacker						: BOOL;
	bAggregationWithoutCamera					: BOOL;
	bOrcaExist										: BOOL;

(*Commisioning settings*)
	bDisableOuterReject						: BOOL;	(*Disable any outer reject - just for commisioning*)
	bDisableCaseReject						: BOOL;	(*Disable any case reject - just for commisioning*)
	bOuterRejectWithHighSignal				: BOOL;
	bCaseRejectWithHighSignal				: BOOL;

(* Device Settings*)
	bUPSExist										: BOOL;
	bUPSImmediateShutdown						: BOOL := FALSE;		(*Option to control immediate shutdown on power loss*)

	bApplyLabelInPassthrough					: BOOL;
	bDisableApplyLabel						: BOOL;
	bPrinterHighSpeedEnable					: BOOL;
	bEANValidationEnable						: BOOL;

	bPrintSignalFromPLC						: BOOL;
	bEnableResendCommand					: BOOL;

(*******************************************************************************************************************************************************)
(********************************************************Numercis******************************************************************************)
(*******************************************************************************************************************************************************)
(*Line system type set up*)
	nPackAggregationMode						: INT := 0; (* 0 -NOPACKAGGREGATION, 1 -STRUCTURALAGGREGATION (PAOL), 2 -STRUCTURALAGGREGATION (2CAM),  3 - LINEARAGGREGATION (PLAS), 4 - NCWAGGREGATION (PLAS + INTERIM)*)
	nOuterAggregationMode						: INT := 0; (* 0 - SYNCHROCONFIRMATION, 1 - SHIFTCONFIRMATION, 2 -SFLXNOCONFIRMATION, 3 - SFLXWITHCONFIRMATION, 4 - LASERPRINTLABEL*)
	nAutomationMode								: INT := 0; (* 0 - EXTERNAL, 1 - CML, 2 - LARS, 3 - SIDEFLEX *)

(* Consecutive rejects counter*)
	nConsecutivePackRejects						: UINT := 3;
	nConsecutivePackConfirmationMissing		: UINT := 3;
	nConsecutiveOCVMissing						: UINT := 3;
	nConsecutiveIntermediateNoRead				: UINT := 3;
	nConsecutiveOuterRejects						: UINT := 3;
	nConsecutiveCaseContentMissing				: UINT := 3;
	nConsecutiveCaseRejects						: UINT := 3;

(*Archive settings*)
	nMaximumArchiveAge							: INT := 28;		(*Max archive age in days*)
	nMaximumArchiveFiles						: INT := 100;

	nMaximumOCVFiles							: INT := 5000;
	nMaximumOACFiles							: INT := 1000;
	nMaximumErrorFiles							: INT := 100;

(* HMI settings*)
	nWarningLevelPack							: REAL := 99.95;
	nAlarmLevelPack								: REAL := 99.9;
	nWarningLevelOuter							: REAL := 99.5;
	nAlarmLevelOuter								: REAL := 99.0;
	nWarningLevelCase							: REAL := 99.5;
	nAlarmLevelCase								: REAL := 95.0;

	tPassthroughDisableDelay						: TIME := t#2s;
(*SequenceTimeOut*)
	tPackMasterListTimeout						: TIME := t#250ms;
	tPackAgreggationTimeout						: TIME := t#500ms;
	tPackConfirmationTimeout					: TIME := t#500ms;
	tInterimTimeout								: TIME := T#500ms;
	tOuterValidationTimeout						: TIME := t#750ms;
(*Sensors Timeouts*)
	tRejectSensorTimeout							: TIME := T#10s;
	tRowCompleteSignalTimeOut					: TIME := t#25s;
	tLayerCompleteSignalTimeOut					: TIME := t#25s;
	tIntermediatePushSignalTimeOut				: TIME := t#25s;
	tCaseCompleteSignalTimeOut					: TIME := t#25s;
	tDischargeSignalTimeOut						: TIME := t#25s;
	tCaseLabelValidationSignalTimeOut			: TIME := t#25s;
	tCaseRejectTimeOut							: TIME := t#60s;

(*Pack*)
	nAggregationUnitLightingIntensityTop		: INT := 100;		(*to be removed and replaced with camera config*)
	nAggregationUnitLightingIntensity			: INT := 100;				(*to be removed and replaced with camera config*)
	tLightboxLensAirFrequency					: TIME := t#3h;
	tLightboxLensAirBlowDuration				: TIME := t#10s;
	nClearPMLIndex								: INT;
	nClearPMLRecords								: INT;
	stPackAgregationCameraOffset				: ST_PACK_TriggerOffset;	(*Used for SFLX 2 Cam aggregation*)
	stPackCamera01Offset							: ST_PACK_TriggerOffset;	(*Used for SFLX 2 Cam aggregation*)
	stPackCamera02Offset							: ST_PACK_TriggerOffset;	(*Used for SFLX 2 Cam aggregation*)

	nConfirmationPackCode1						: INT := 1;
	nConfirmationPackCode2						: INT := 2;
	nPacksPerStack								: UINT := 5;
	nMaxOutersBuffer								: UINT := 1; 		(*Maximum number of outers that can be processes at one time allowing for camera buffers - can be set higher if camera sequence max buffer is fixed!*)
	tBufferDelayTime								: TIME := t#200ms; 		(*Adjust this time so each outer stops for a moment before the first infeed camera sensor in order to avoid out of sync errors*)
	nCheckStatusOCV								: BYTE := 2;
	nExpectedValidationDepth						: INT := 1;
	nInterimQueueIndex							: INT :=1;

(*Outer*)
	nOutersPerRow									: INT := 5;
	tTwoOutersOnRejectConv						: TIME := T#500ms;
	nMasterListNumbersWarning					: INT := 5;
	nAuxRowCount								: INT := 2;
	nAggregationQueueIndex						: INT := 0;
	tInspectionDelay								: TIME := t#30ms;

(* Case*)
	nCaseQueueLength							: INT := 3;
	nCaseContentBuffer							: INT;

(*Device*)
	tUPSShutdownDelay							: TIME := t#30s;		(*Default grace period for NT_Shutdown FB*)

(*******************************************************************************************************************************************************)
(********************************************************Devices******************************************************************************)
(*******************************************************************************************************************************************************)
(*Camera - IP/Port settings for All scanners used in EUCA-TPD  arrays with up to 6 scanners per array *)
	aCameraSettings							: ARRAY [1..cMAX_CAMERA_NUMBER] OF ST_SCANNER_Config;

(*Printers*)
	aPrinterSettings							: ARRAY [1..cMAX_PRINTER_NUMBER] OF ST_PRINTER_Config;

(*Hand Scanners*)
	aHandScannersConfig						: ARRAY [1..cMAX_HAND_SCANNERS] OF ST_SCANNER_HoneywellConfig;
	aHoneywellCtrl								: ARRAY [1..cMAX_HAND_SCANNERS] OF ST_SCANNER_HoneywellCtrl;
	stUSBScannerConfig						: ST_SCANNER_USBConfig;

(* Profinet drives *)
	aProfiNetMaster							: ARRAY [1..cMAX_PROFINET_MASTERS]  OF  ST_ProfinetMasterConfig; (* EL6631 *)
	aProfiNetDrive								: ARRAY [1..cMAX_PROFINET_DRIVES]  OF ST_ProfinetDrive; (*config for individual drives *)

(*MC2 drives*)
	aAxisConfig								: ARRAY [1..cMAX_MC2_DRIVES] OF ST_AXIS_Config;

(* Analog drive*)
	stPackSeparator							: ST_AnalogDrive;

(*Cylinders*)
	aCylinderConfig							: ARRAY [1..cMAX_CYLINDERS] OF ST_CYLINDER_Config;

(* CAMS  *)
	(*aAFS50camConfig						: ARRAY [1.. cMAX_CAMS] OF ST_AFS60_Config;*)

(*Database*)
	(*stDBConfig								: ST_DB_Config;*)

(*******************************************************************************************************************************************************)
(********************************************************Single IO******************************************************************************)
(*******************************************************************************************************************************************************)
(*Single Input Config*)
	st_I_TransferCoveyorDoorGuard1			: ST_IO2_SingleInputCtrl:=			(eTypeInput:=E_IO2_Type.NO,		tTimeOnFilter:=t#100ms, 		tTimeOffFilter:=t#10ms, 	sInputName:='Transfer Coveyor Door Guard 1' );	(**)
	st_I_TransferCoveyorDoorGuard2			: ST_IO2_SingleInputCtrl:=			(eTypeInput:=E_IO2_Type.NO,		tTimeOnFilter:=t#100ms, 		tTimeOffFilter:=t#10ms, 	sInputName:='Transfer Coveyor Door Guard 2' );	(**)

	st_I_DoorOpenZone1					: ST_IO2_SingleInputCtrl:=			(eTypeInput:=E_IO2_Type.NO,		tTimeOnFilter:=t#100ms, 		tTimeOffFilter:=t#10ms, 	sInputName:='Door Open Zone 1' );	(**)
	st_I_DoorOpenZone2					: ST_IO2_SingleInputCtrl:=			(eTypeInput:=E_IO2_Type.NO,		tTimeOnFilter:=t#100ms, 		tTimeOffFilter:=t#10ms, 	sInputName:='Door Open Zone 2' );	(**)

	st_I_AuxRowCompleteSesnor			: ST_IO2_SingleInputCtrl:=			(eTypeInput:=E_IO2_Type.NO,		tTimeOnFilter:=t#10ms, 		tTimeOffFilter:=t#10ms, 	sInputName:='Aux Row Complete' );	(**)
	st_I_CaseRejectedByCasePacker		: ST_IO2_SingleInputCtrl:=			(eTypeInput:=E_IO2_Type.NO,		tTimeOnFilter:=t#10ms, 		tTimeOffFilter:=t#10ms, 	sInputName:='Case Rejected By Casepacker' );	(**)

	st_I_PreMachineAutoRun				: ST_IO2_SingleInputCtrl:=			(eTypeInput:=E_IO2_Type.NO,		tTimeOnFilter:=t#100ms, 		tTimeOffFilter:=t#0ms, 	sInputName:='PreMachine AutoRun' );	(**)
	st_I_CasePackerAutoRun				: ST_IO2_SingleInputCtrl:=			(eTypeInput:=E_IO2_Type.NO,		tTimeOnFilter:=t#100ms, 		tTimeOffFilter:=t#0ms, 	sInputName:='Casepacker AutoRun' );	(**)

	st_I_QAButtonRejectOuter				: ST_IO2_SingleInputCtrl:=			(eTypeInput:=E_IO2_Type.NO,		tTimeOnFilter:=t#100ms, 		tTimeOffFilter:=t#0ms, 	sInputName:='QA Button Reject Outer' );	(**)
	st_I_OuterAtRejectStation				: ST_IO2_SingleInputCtrl:=			(eTypeInput:=E_IO2_Type.NO,		tTimeOnFilter:=t#1000ms, 		tTimeOffFilter:=t#0ms, 	sInputName:='Outer At Reject Station' );	(**)
	st_I_OuterRejectConfirm				: ST_IO2_SingleInputCtrl:=			(eTypeInput:=E_IO2_Type.NO,		tTimeOnFilter:=t#1000ms, 		tTimeOffFilter:=t#0ms, 	sInputName:='Outer Reject Confirm' );	(**)
	st_I_RejectBinFull						: ST_IO2_SingleInputCtrl:=			(eTypeInput:=E_IO2_Type.NO,		tTimeOnFilter:=t#100ms, 		tTimeOffFilter:=t#0ms, 	sInputName:='Reject Bin Full' );	(**)

	st_I_EUCABuildBackPreMachine			: ST_IO2_SingleInputCtrl:=			(eTypeInput:=E_IO2_Type.NO,		tTimeOnFilter:=t#1000ms, 		tTimeOffFilter:=t#0ms, 	sInputName:='EUCA Buildback Sensor' );	(**)
	st_I_EUCAExitBlocked						: ST_IO2_SingleInputCtrl:=			(eTypeInput:=E_IO2_Type.NO,		tTimeOnFilter:=t#1000ms, 		tTimeOffFilter:=t#0ms, 	sInputName:='EUCA Exit Blocked Sensor' );	(**)

	st_I_OuterAtSystemInfeed					: ST_IO2_SingleInputCtrl:=			(eTypeInput:=E_IO2_Type.NO,		tTimeOnFilter:=t#1000ms, 		tTimeOffFilter:=t#0ms, 	sInputName:='Outer At System Infeed Sensor' );	(**)
	st_I_OuterAtAdditionalConv				: ST_IO2_SingleInputCtrl:=			(eTypeInput:=E_IO2_Type.NO,		tTimeOnFilter:=t#1000ms, 		tTimeOffFilter:=t#0ms, 	sInputName:='Outer At Additional Conv Sensor' );	(**)

	st_I_TransferConveyorPlugConnected		: ST_IO2_SingleInputCtrl:=			(eTypeInput:=E_IO2_Type.NO,		tTimeOnFilter:=t#100ms, 		tTimeOffFilter:=t#100ms, 	sInputName:='Transfer Conveyor Plug Connected' );	(**)
	st_I_OutfeedConveyorPlugConnected		: ST_IO2_SingleInputCtrl:=			(eTypeInput:=E_IO2_Type.NO,		tTimeOnFilter:=t#100ms, 		tTimeOffFilter:=t#100ms, 	sInputName:='Outfeed Conveyor Plug Connected' );	(**)
	st_I_AdditionalConveyorPlugConnected	: ST_IO2_SingleInputCtrl:=			(eTypeInput:=E_IO2_Type.NO,		tTimeOnFilter:=t#100ms, 		tTimeOffFilter:=t#100ms, 	sInputName:='Outfeed Conveyor Plug Connected' );	(**)

(*Single Input Config for camera triggers*)
	st_I_Camera01						: ST_IO2_SingleInputCtrl:=			(eTypeInput:=E_IO2_Type.NO,		tTimeOnFilter:=t#6ms, 		tTimeOffFilter:=t#20ms, 	sInputName:='Camera 01' );	(**)
	st_I_Camera02						: ST_IO2_SingleInputCtrl:=			(eTypeInput:=E_IO2_Type.NO,		tTimeOnFilter:=t#6ms, 		tTimeOffFilter:=t#20ms, 	sInputName:='Camera 02' );	(**)
	st_I_Camera03						: ST_IO2_SingleInputCtrl:=			(eTypeInput:=E_IO2_Type.NO,		tTimeOnFilter:=t#6ms, 		tTimeOffFilter:=t#20ms, 	sInputName:='Camera 03' );	(**)
	st_I_Camera04						: ST_IO2_SingleInputCtrl:=			(eTypeInput:=E_IO2_Type.NO,		tTimeOnFilter:=t#10ms, 		tTimeOffFilter:=t#0ms, 	sInputName:='Camera 04' );	(**)
	st_I_Camera05						: ST_IO2_SingleInputCtrl:=			(eTypeInput:=E_IO2_Type.NO,		tTimeOnFilter:=t#10ms, 		tTimeOffFilter:=t#0ms, 	sInputName:='Camera 05' );	(**)
	st_I_Camera06						: ST_IO2_SingleInputCtrl:=			(eTypeInput:=E_IO2_Type.NO,		tTimeOnFilter:=t#10ms, 		tTimeOffFilter:=t#0ms, 	sInputName:='Camera 06' );	(**)
	st_I_Camera07						: ST_IO2_SingleInputCtrl:=			(eTypeInput:=E_IO2_Type.NO,		tTimeOnFilter:=t#10ms, 		tTimeOffFilter:=t#0ms, 	sInputName:='Camera 07' );	(**)
	st_I_Camera08						: ST_IO2_SingleInputCtrl:=			(eTypeInput:=E_IO2_Type.NO,		tTimeOnFilter:=t#10ms, 		tTimeOffFilter:=t#0ms, 	sInputName:='Camera 08' );	(**)
	st_I_Camera09						: ST_IO2_SingleInputCtrl:=			(eTypeInput:=E_IO2_Type.NO,		tTimeOnFilter:=t#10ms, 		tTimeOffFilter:=t#0ms, 	sInputName:='Camera 09' );	(**)
	st_I_Camera10						: ST_IO2_SingleInputCtrl:=			(eTypeInput:=E_IO2_Type.NO,		tTimeOnFilter:=t#10ms, 		tTimeOffFilter:=t#0ms, 	sInputName:='Camera 10' );	(**)
	st_I_Camera11						: ST_IO2_SingleInputCtrl:=			(eTypeInput:=E_IO2_Type.NO,		tTimeOnFilter:=t#10ms, 		tTimeOffFilter:=t#0ms, 	sInputName:='Camera 11' );	(**)
	st_I_Camera12						: ST_IO2_SingleInputCtrl:=			(eTypeInput:=E_IO2_Type.NO,		tTimeOnFilter:=t#10ms, 		tTimeOffFilter:=t#0ms, 	sInputName:='Camera 12' );	(**)

(*METS Cylinders Filtered Inputs *)
	st_I_ClampCylinderExtended		: ST_IO2_SingleInputCtrl:=			(eTypeInput:=E_IO2_Type.NO,		tTimeOnFilter:=t#10ms, 		tTimeOffFilter:=t#0ms, 	sInputName:='Clamp Cylinder Extended' );	(**)
	st_I_ClampCylinderRetracted		: ST_IO2_SingleInputCtrl:=			(eTypeInput:=E_IO2_Type.NO,		tTimeOnFilter:=t#10ms, 		tTimeOffFilter:=t#0ms, 	sInputName:='Clamp Cylinder Retracted' );	(**)

	st_I_GateCylinderExtended		: ST_IO2_SingleInputCtrl:=			(eTypeInput:=E_IO2_Type.NO,		tTimeOnFilter:=t#10ms, 		tTimeOffFilter:=t#0ms, 	sInputName:='Gate Cylinder Extended' );	(**)
	st_I_GateCylinderRetracted 		: ST_IO2_SingleInputCtrl:=			(eTypeInput:=E_IO2_Type.NO,		tTimeOnFilter:=t#10ms, 		tTimeOffFilter:=t#0ms, 	sInputName:='Gate Cylinder Retracted' );	(**)

	st_I_RejectCylinderExtended		: ST_IO2_SingleInputCtrl:=			(eTypeInput:=E_IO2_Type.NO,		tTimeOnFilter:=t#10ms, 		tTimeOffFilter:=t#0ms, 	sInputName:='Reject Cylinder Extended' );	(**)
	st_I_RejectCylinderRetracted 		: ST_IO2_SingleInputCtrl:=			(eTypeInput:=E_IO2_Type.NO,		tTimeOnFilter:=t#10ms, 		tTimeOffFilter:=t#0ms, 	sInputName:='Reject Cylinder Retracted' );	(**)

	st_I_AdditionalRejectCylinderExtended		: ST_IO2_SingleInputCtrl:=			(eTypeInput:=E_IO2_Type.NO,		tTimeOnFilter:=t#10ms, 		tTimeOffFilter:=t#0ms, 	sInputName:='Reject Cylinder Extended' );	(**)
	st_I_AdditionalRejectCylinderRetracted 		: ST_IO2_SingleInputCtrl:=			(eTypeInput:=E_IO2_Type.NO,		tTimeOnFilter:=t#10ms, 		tTimeOffFilter:=t#0ms, 	sInputName:='Reject Cylinder Retracted' );	(**)

	st_I_FirstPusherCylinderExtended		: ST_IO2_SingleInputCtrl:=			(eTypeInput:=E_IO2_Type.NO,		tTimeOnFilter:=t#10ms, 		tTimeOffFilter:=t#0ms, 	sInputName:='Reject Cylinder Extended' );	(**)
	st_I_FirstPusherCylinderRetracted 		: ST_IO2_SingleInputCtrl:=			(eTypeInput:=E_IO2_Type.NO,		tTimeOnFilter:=t#10ms, 		tTimeOffFilter:=t#0ms, 	sInputName:='Reject Cylinder Retracted' );	(**)

	st_I_SecondPusherCylinderExtended		: ST_IO2_SingleInputCtrl:=			(eTypeInput:=E_IO2_Type.NO,		tTimeOnFilter:=t#10ms, 		tTimeOffFilter:=t#0ms, 	sInputName:='Reject Cylinder Extended' );	(**)
	st_I_SecondPusherCylinderRetracted 		: ST_IO2_SingleInputCtrl:=			(eTypeInput:=E_IO2_Type.NO,		tTimeOnFilter:=t#10ms, 		tTimeOffFilter:=t#0ms, 	sInputName:='Reject Cylinder Retracted' );	(**)

(*METS Labellers Filtered Inputs *)
	st_I_Labeller1InPosition					: ST_IO2_SingleInputCtrl:=			(eTypeInput:=E_IO2_Type.NO,		tTimeOnFilter:=t#10ms, 		tTimeOffFilter:=t#0ms, 	sInputName:='Labeller1 In Position' );	(**)
	st_I_Labeller1OuterAtLabeller				: ST_IO2_SingleInputCtrl:=			(eTypeInput:=E_IO2_Type.NO,		tTimeOnFilter:=t#10ms, 		tTimeOffFilter:=t#0ms, 	sInputName:='Labeller1 Outer At Labeller' );	(**)
	tLabeller1OuterAtLabellerTimeLatch		: TIME := t#200ms; (*Variable used separately to keep one standard with HMI user controls for Single Inputs*)

	st_I_Labeller1Ready						: ST_IO2_SingleInputCtrl:=			(eTypeInput:=E_IO2_Type.NO,		tTimeOnFilter:=t#10ms, 		tTimeOffFilter:=t#0ms, 	sInputName:='Labeller1 Ready' );	(**)
	st_I_Labeller1DataReady					: ST_IO2_SingleInputCtrl:=			(eTypeInput:=E_IO2_Type.NO,		tTimeOnFilter:=t#10ms, 		tTimeOffFilter:=t#0ms, 	sInputName:='Labeller1 Data Ready' );	(**)
	st_I_Labeller1HomePosition				: ST_IO2_SingleInputCtrl:=			(eTypeInput:=E_IO2_Type.NO,		tTimeOnFilter:=t#10ms, 		tTimeOffFilter:=t#0ms, 	sInputName:='Labeller1 Home Position' );	(**)
	st_I_Labeller1LabelPrinted					: ST_IO2_SingleInputCtrl:=			(eTypeInput:=E_IO2_Type.NO,		tTimeOnFilter:=t#10ms, 		tTimeOffFilter:=t#0ms, 	sInputName:='Labeller1 Label Printed' );	(**)
	st_I_Labeller1ReadyToApply				: ST_IO2_SingleInputCtrl:=			(eTypeInput:=E_IO2_Type.NO,		tTimeOnFilter:=t#10ms, 		tTimeOffFilter:=t#0ms, 	sInputName:='Labeller1 Ready To Apply' );	(**)
	st_I_Labeller1ApplyDone					: ST_IO2_SingleInputCtrl:=			(eTypeInput:=E_IO2_Type.NO,		tTimeOnFilter:=t#10ms, 		tTimeOffFilter:=t#0ms, 	sInputName:='Labeller1 Apply Done' );	(**)
	st_I_Labeller1SummaryWarning			: ST_IO2_SingleInputCtrl:=			(eTypeInput:=E_IO2_Type.NO,		tTimeOnFilter:=t#10ms, 		tTimeOffFilter:=t#0ms, 	sInputName:='Labeller1 Summary Warning' );	(**)
	st_I_Labeller1Error							: ST_IO2_SingleInputCtrl:=			(eTypeInput:=E_IO2_Type.NO,		tTimeOnFilter:=t#10ms, 		tTimeOffFilter:=t#0ms, 	sInputName:='Labeller1 Error' );	(**)


	st_I_Labeller2InPosition					: ST_IO2_SingleInputCtrl:=			(eTypeInput:=E_IO2_Type.NO,		tTimeOnFilter:=t#10ms, 		tTimeOffFilter:=t#0ms, 	sInputName:='Labeller2 In Position' );	(**)
	st_I_Labeller2OuterAtLabeller				: ST_IO2_SingleInputCtrl:=			(eTypeInput:=E_IO2_Type.NO,		tTimeOnFilter:=t#10ms, 		tTimeOffFilter:=t#0ms, 	sInputName:='Labeller2 Outer At Labeller' );	(**)
	tLabeller2OuterAtLabellerTimeLatch		: TIME := t#40ms; (*Variable used separately to keep one standard with HMI user controls for Single Inputs*)

	st_I_Labeller2Ready						: ST_IO2_SingleInputCtrl:=			(eTypeInput:=E_IO2_Type.NO,		tTimeOnFilter:=t#10ms, 		tTimeOffFilter:=t#0ms, 	sInputName:='Labeller2 Ready' );	(**)
	st_I_Labeller2DataReady					: ST_IO2_SingleInputCtrl:=			(eTypeInput:=E_IO2_Type.NO,		tTimeOnFilter:=t#10ms, 		tTimeOffFilter:=t#0ms, 	sInputName:='Labeller2 Data Ready' );	(**)
	st_I_Labeller2HomePosition				: ST_IO2_SingleInputCtrl:=			(eTypeInput:=E_IO2_Type.NO,		tTimeOnFilter:=t#10ms, 		tTimeOffFilter:=t#0ms, 	sInputName:='Labeller2 Home Position' );	(**)
	st_I_Labeller2LabelPrinted					: ST_IO2_SingleInputCtrl:=			(eTypeInput:=E_IO2_Type.NO,		tTimeOnFilter:=t#10ms, 		tTimeOffFilter:=t#0ms, 	sInputName:='Labeller2 Label Printed' );	(**)
	st_I_Labeller2ReadyToApply				: ST_IO2_SingleInputCtrl:=			(eTypeInput:=E_IO2_Type.NO,		tTimeOnFilter:=t#10ms, 		tTimeOffFilter:=t#0ms, 	sInputName:='Labeller2 Ready To Apply' );	(**)
	st_I_Labeller2ApplyDone					: ST_IO2_SingleInputCtrl:=			(eTypeInput:=E_IO2_Type.NO,		tTimeOnFilter:=t#10ms, 		tTimeOffFilter:=t#0ms, 	sInputName:='Labeller2 Apply Done' );	(**)
	st_I_Labeller2SummaryWarning			: ST_IO2_SingleInputCtrl:=			(eTypeInput:=E_IO2_Type.NO,		tTimeOnFilter:=t#10ms, 		tTimeOffFilter:=t#0ms, 	sInputName:='Labeller2 Summar yWarning' );	(**)
	st_I_Labeller2Error							: ST_IO2_SingleInputCtrl:=			(eTypeInput:=E_IO2_Type.NO,		tTimeOnFilter:=t#10ms, 		tTimeOffFilter:=t#0ms, 	sInputName:='Labeller2 Error' );	(**)

(*METS SADDLE (Gating&Reject System) Filtered Inputs  FB***************************************************************************************************************)
	st_I_OuterAtClamp					: ST_IO2_SingleInputCtrl:=			(eTypeInput:=E_IO2_Type.NO,		tTimeOnFilter:=t#100ms, 		tTimeOffFilter:=t#100ms, 		sInputName:='Outer At Clamp');	(**)
	st_I_OuterAtLabelGate				: ST_IO2_SingleInputCtrl:=			(eTypeInput:=E_IO2_Type.NO,		tTimeOnFilter:=t#100ms, 		tTimeOffFilter:=t#100ms, 		sInputName:='Outer At Label Gate');	(**)
	st_I_GateClear						: ST_IO2_SingleInputCtrl:=			(eTypeInput:=E_IO2_Type.NO,		tTimeOnFilter:=t#100ms, 		tTimeOffFilter:=t#100ms, 		sInputName:='Gate Clear');	(**)
	st_I_GateImpact					: ST_IO2_SingleInputCtrl:=			(eTypeInput:=E_IO2_Type.NO,		tTimeOnFilter:=t#100ms, 		tTimeOffFilter:=t#100ms, 		sInputName:='Gate Impact');	(**)

(* Single Inputs for METS CML*)
	st_I_RotaryTransferPackAtStopPlate		: ST_IO2_SingleInputCtrl:=			(eTypeInput:=E_IO2_Type.NO,		tTimeOnFilter:=t#1000ms, 		tTimeOffFilter:=t#0ms, 	sInputName:='Rotary Transfer Outer At Stop Plate');	(**)
	st_I_RotaryTransferTorqueLimiter			: ST_IO2_SingleInputCtrl:=			(eTypeInput:=E_IO2_Type.NO,		tTimeOnFilter:=t#1000ms, 		tTimeOffFilter:=t#0ms, 	sInputName:='Rotary Transfer Torque Limiter');	(**)
	st_I_RotaryTransferDelayStop1			: ST_IO2_SingleInputCtrl:=			(eTypeInput:=E_IO2_Type.NO,		tTimeOnFilter:=t#1000ms, 		tTimeOffFilter:=t#0ms, 	sInputName:='Rotary Transfer Delay Stop1');	(**)
	st_I_RotaryTransferDelayStop2			: ST_IO2_SingleInputCtrl:=			(eTypeInput:=E_IO2_Type.NO,		tTimeOnFilter:=t#1000ms, 		tTimeOffFilter:=t#0ms, 	sInputName:='Rotary Transfer Delay Stop2');	(**)
	st_I_ConveyorIndexContact				: ST_IO2_SingleInputCtrl:=			(eTypeInput:=E_IO2_Type.NO,		tTimeOnFilter:=t#50ms, 		tTimeOffFilter:=t#50s, 	sInputName:='Infeed Conveyor Start');	(**)
	st_I_Guard4ElectricalBoxInPosition		: ST_IO2_SingleInputCtrl:=			(eTypeInput:=E_IO2_Type.NC,		tTimeOnFilter:=t#50ms, 		tTimeOffFilter:=t#50s, 	sInputName:='Electrical Box In Position Sensor');	(**)

(* Single Inputs for METS Manual Machine*)
	st_I_InfeedConveyorStart				: ST_IO2_SingleInputCtrl:=			(eTypeInput:=E_IO2_Type.NO,		tTimeOnFilter:=t#1000ms, 		tTimeOffFilter:=t#0ms, 	sInputName:='Infeed Conveyor Start');	(**)
	st_I_RejectChuteExitBlocked			: ST_IO2_SingleInputCtrl:=			(eTypeInput:=E_IO2_Type.NO,		tTimeOnFilter:=t#1000ms, 		tTimeOffFilter:=t#0ms, 	sInputName:='Reject Chute Blocked');	(**)

(* Single Inputs for METS SFLX Machine*)
	st_I_OuterInfeedJam						: ST_IO2_SingleInputCtrl:=			(eTypeInput:=E_IO2_Type.NO,		tTimeOnFilter:=t#1000ms, 		tTimeOffFilter:=t#0ms, 	sInputName:='Outer Infeed Jam' );	(**)
	(*st_I_PackAggregationCameraTrigger		: ST_IO2_SingleInputCtrl:=			(eTypeInput:=E_IO2_Type.NO,		tTimeOnFilter:=t#1000ms, 		tTimeOffFilter:=t#0ms, 	sInputName:='Pack Aggregation Camera Trigger');*)	(**)
	st_I_OutfeedConveyorStart				: ST_IO2_SingleInputCtrl:=			(eTypeInput:=E_IO2_Type.NO,		tTimeOnFilter:=t#1000ms, 		tTimeOffFilter:=t#0ms, 	sInputName:='Outfeed Conveyor Start');	(**)
	st_I_RejectConfirmationNCW				: ST_IO2_SingleInputCtrl:=			(eTypeInput:=E_IO2_Type.NO,		tTimeOnFilter:=t#1000ms, 		tTimeOffFilter:=t#0ms, 	sInputName:='Reject Confirmation NCW');	(**)
	st_I_RejectBinFullNCW						: ST_IO2_SingleInputCtrl:=			(eTypeInput:=E_IO2_Type.NO,		tTimeOnFilter:=t#1000ms, 		tTimeOffFilter:=t#0ms, 	sInputName:='Reject Bin Full NCW');	(**)
	st_I_OuterAtTransferReject				: ST_IO2_SingleInputCtrl:=			(eTypeInput:=E_IO2_Type.NO,		tTimeOnFilter:=t#1000ms, 		tTimeOffFilter:=t#0ms, 	sInputName:='Outer At Transfer Reject');	(**)
	st_I_OuterAtSideFlexExit					: ST_IO2_SingleInputCtrl:=			(eTypeInput:=E_IO2_Type.NO,		tTimeOnFilter:=t#1000ms, 		tTimeOffFilter:=t#0ms, 	sInputName:='Outer At Side Flex Exit');	(**)
	st_I_OuterAtPostMachineInfeed			: ST_IO2_SingleInputCtrl:=			(eTypeInput:=E_IO2_Type.NO,		tTimeOnFilter:=t#1000ms, 		tTimeOffFilter:=t#0ms, 	sInputName:='Outer At PostMachine Infeed');	(**)

	st_I_Guard1FlexInfeedDoor				: ST_IO2_SingleInputCtrl:=			(eTypeInput:=E_IO2_Type.NC,		tTimeOnFilter:=t#1000ms, 		tTimeOffFilter:=t#0ms, 	sInputName:='Guard 1 Flex Infeed Door');	(**)
	st_I_Guard3FlexRHDoor					: ST_IO2_SingleInputCtrl:=			(eTypeInput:=E_IO2_Type.NO,		tTimeOnFilter:=t#200ms, 		tTimeOffFilter:=t#200ms, 	sInputName:='Guard 3 Flex RH Door');	(**)
	st_I_Guard4FlexPrinterDoor				: ST_IO2_SingleInputCtrl:=			(eTypeInput:=E_IO2_Type.NO,		tTimeOnFilter:=t#200ms, 		tTimeOffFilter:=t#200ms, 	sInputName:='Guard 4 Flex Printer Door');	(**)
	st_I_Guard5FlexLHDoor					: ST_IO2_SingleInputCtrl:=			(eTypeInput:=E_IO2_Type.NO,		tTimeOnFilter:=t#200ms, 		tTimeOffFilter:=t#200ms, 	sInputName:='Guard 5 Flex LH Door	');	(**)

(*Single Input for PACAN*)
(*	st_I_StackerArmAtBackwardPosition	: ST_IO2_SingleInputCtrl:=			(eTypeInput:=E_IO2_Type.NO,		tTimeOnFilter:=t#10ms, 		tTimeOffFilter:=t#0ms, 	sInputName:='Stacker Arm At Backward Position');	(**)
	st_I_StackerArmInTopPosition			: ST_IO2_SingleInputCtrl:=			(eTypeInput:=E_IO2_Type.NO,		tTimeOnFilter:=t#10ms, 		tTimeOffFilter:=t#0ms, 	sInputName:='Stacker Arm In Top Position');	(**)
	st_I_StackPresentSensor1				: ST_IO2_SingleInputCtrl:=			(eTypeInput:=E_IO2_Type.NO,		tTimeOnFilter:=t#10ms, 		tTimeOffFilter:=t#0ms, 	sInputName:='Stack Present Sensor1');	(**)
	st_I_StackPresentSensor2				: ST_IO2_SingleInputCtrl:=			(eTypeInput:=E_IO2_Type.NO,		tTimeOnFilter:=t#10ms, 		tTimeOffFilter:=t#0ms, 	sInputName:='Stack Present Sensor2');	(**)
	st_I_StackerTransferPusher			: ST_IO2_SingleInputCtrl:=			(eTypeInput:=E_IO2_Type.NO,		tTimeOnFilter:=t#10ms, 		tTimeOffFilter:=t#0ms, 	sInputName:='Stacker Transfer Pusher');	(**)
	st_I_StackerTransferComplete			: ST_IO2_SingleInputCtrl:=			(eTypeInput:=E_IO2_Type.NO,		tTimeOnFilter:=t#10ms, 		tTimeOffFilter:=t#0ms, 	sInputName:='Stacker Transfer Complete');	(**)
	st_I_OuterAtPACANRejectStation		: ST_IO2_SingleInputCtrl:=			(eTypeInput:=E_IO2_Type.NO,		tTimeOnFilter:=t#100ms, 		tTimeOffFilter:=t#100ms, 	sInputName:='Outer At PACAN Reject Station');	(**)
*)
(*Single Input for PAOL*)
	st_I_TPDExitBlockedSensor			: ST_IO2_SingleInputCtrl:=			(eTypeInput:=E_IO2_Type.NO,		tTimeOnFilter:=t#100ms, 		tTimeOffFilter:=t#0ms, 	sInputName:='PAOL Exit Blocked Sensor');	(**)
	st_I_PreMachineBuildBackSensor		: ST_IO2_SingleInputCtrl:=			(eTypeInput:=E_IO2_Type.NO,		tTimeOnFilter:=t#100ms, 		tTimeOffFilter:=t#0ms, 	sInputName:='PAOL Buildback Sensor');	(**)
	st_I_PackAggregCameraRigSensor		: ST_IO2_SingleInputCtrl:=			(eTypeInput:=E_IO2_Type.NO,		tTimeOnFilter:=t#6ms, 		tTimeOffFilter:=t#6ms, 	sInputName:='Pack Aggreg Camera Rig Sensor');	(**)

(*Single Input for PLAS*)
	st_I_MasterlistDoorGuard1				: ST_IO2_SingleInputCtrl:=			(eTypeInput:=E_IO2_Type.NC,		tTimeOnFilter:=t#50ms, 		tTimeOffFilter:=t#50ms, 	sInputName:='Masterlist Door Guard1');	(**)
	st_I_MasterlistDoorGuard2				: ST_IO2_SingleInputCtrl:=			(eTypeInput:=E_IO2_Type.NC,		tTimeOnFilter:=t#50ms, 		tTimeOffFilter:=t#50ms, 	sInputName:='Masterlist Door Guard2');	(**)
	st_I_MasterlistDoorGuard3				: ST_IO2_SingleInputCtrl:=			(eTypeInput:=E_IO2_Type.NC,		tTimeOnFilter:=t#50ms, 		tTimeOffFilter:=t#50ms, 	sInputName:='Masterlist Door Guard3');	(**)

	st_I_OuterBrushOpen						: ST_IO2_SingleInputCtrl:=			(eTypeInput:=E_IO2_Type.NC,		tTimeOnFilter:=t#50ms, 		tTimeOffFilter:=t#50ms, 	sInputName:='Outer Brush Open');	(**)
	st_I_PackAggregationDoorGuard1			: ST_IO2_SingleInputCtrl:=			(eTypeInput:=E_IO2_Type.NC,		tTimeOnFilter:=t#50ms, 		tTimeOffFilter:=t#50ms, 	sInputName:='Pack Aggregation Door Guard1');	(**)
	st_I_PackAggregationDoorGuard2			: ST_IO2_SingleInputCtrl:=			(eTypeInput:=E_IO2_Type.NC,		tTimeOnFilter:=t#50ms, 		tTimeOffFilter:=t#50ms, 	sInputName:='Pack Aggregation Door Guard2');	(**)

	st_I_WrapperDoorGuard1					:  ST_IO2_SingleInputCtrl:=			(eTypeInput:=E_IO2_Type.NC,		tTimeOnFilter:=t#50ms, 		tTimeOffFilter:=t#50ms, 	sInputName:='Wrapper Door Guard1');	(**)
	st_I_WrapperDoorGuard2					: ST_IO2_SingleInputCtrl:=			(eTypeInput:=E_IO2_Type.NC,		tTimeOnFilter:=t#50ms, 		tTimeOffFilter:=t#50ms, 	sInputName:='Wrapper Door Guard2');	(**)

	st_I_HeatTunelPackReject				: ST_IO2_SingleInputCtrl:=			(eTypeInput:=E_IO2_Type.NO,		tTimeOnFilter:=t#50ms, 		tTimeOffFilter:=t#50ms, 	sInputName:='Heat Tunenel Pack Reject Sensor');	(**)
	st_I_WrapperPackReject				: ST_IO2_SingleInputCtrl:=			(eTypeInput:=E_IO2_Type.NC,		tTimeOnFilter:=t#50ms, 		tTimeOffFilter:=t#50ms, 	sInputName:='Wrapper Pack Reject Sensor');	(**)
	st_I_WrapperPackReject2				: ST_IO2_SingleInputCtrl:=			(eTypeInput:=E_IO2_Type.NC,		tTimeOnFilter:=t#50ms, 		tTimeOffFilter:=t#50ms, 	sInputName:='Wrapper Pack Reject 2 Sensor');	(**)
	st_I_WrapperOuterComplete			: ST_IO2_SingleInputCtrl:=			(eTypeInput:=E_IO2_Type.NC,		tTimeOnFilter:=t#50ms, 		tTimeOffFilter:=t#50ms, 	sInputName:='Wrapper Pushing Arm Sensor');	(**)
	st_I_InhibitIntermediateCamera		: ST_IO2_SingleInputCtrl:=			(eTypeInput:=E_IO2_Type.NC,		tTimeOnFilter:=t#50ms, 		tTimeOffFilter:=t#50ms, 	sInputName:='Inhibit Intermediate Camera');	(**)

(*Single Input for Laser*)
	st_I_CoderReady					: ST_IO2_SingleInputCtrl:=			(eTypeInput:=E_IO2_Type.NO,		tTimeOnFilter:=t#100ms, 		tTimeOffFilter:=t#0ms, 	sInputName:='LASER - Ready');	(**)
	st_I_CoderBusy					: ST_IO2_SingleInputCtrl:=			(eTypeInput:=E_IO2_Type.NO,		tTimeOnFilter:=t#100ms, 		tTimeOffFilter:=t#0ms, 	sInputName:='LASER - Busy');	(**)
	st_I_WrappingMaterialPresent		: ST_IO2_SingleInputCtrl:=			(eTypeInput:=E_IO2_Type.NO,		tTimeOnFilter:=t#100ms, 		tTimeOffFilter:=t#0ms, 	sInputName:='LASER - WrapPresent');	(**)
	st_I_TabKnifeMoving				: ST_IO2_SingleInputCtrl:=			(eTypeInput:=E_IO2_Type.NO,		tTimeOnFilter:=t#100ms, 		tTimeOffFilter:=t#0ms, 	sInputName:='LASER - TabKnife');	(**)


(*******************************************************************************************************************************************************)
(********************************************************Double IO******************************************************************************)
(*******************************************************************************************************************************************************)
(*Double Input Config*)
	st_I_RowComplete						: ST_IO2_DoubleInputCtrl:=		(eInputSource:=E_IO2_InputSource.SENSOR,	sInputName:='Row Complete',
																						eTypeInput1:=E_IO2_Type.NO,		tTimeOnFilter1:=t#0ms,	tTimeOffFilter1	:=t#0ms,	(**)
											 											eTypeInput2:=E_IO2_Type.NO,		tTimeOnFilter2:=t#0ms,	tTimeOffFilter2	:=t#0ms);	(**)
	st_I_LayerComplete					: ST_IO2_DoubleInputCtrl:=		(eInputSource:=E_IO2_InputSource.SENSOR,	sInputName:='Layer Complete',
																						eTypeInput1:=E_IO2_Type.NO,		tTimeOnFilter1:=t#0ms,	tTimeOffFilter1	:=t#0ms,	(**)
											 											eTypeInput2:=E_IO2_Type.NO,		tTimeOnFilter2:=t#0ms,	tTimeOffFilter2	:=t#0ms);	(**)
	st_I_IntermediatePush					: ST_IO2_DoubleInputCtrl:=		(eInputSource:=E_IO2_InputSource.SENSOR,	sInputName:='Intermediate Push',
																						eTypeInput1:=E_IO2_Type.NO,		tTimeOnFilter1:=t#0ms,	tTimeOffFilter1	:=t#0ms,	(**)
											 											eTypeInput2:=E_IO2_Type.NO,		tTimeOnFilter2:=t#0ms,	tTimeOffFilter2	:=t#0ms);	(**)
	st_I_CaseComplete					: ST_IO2_DoubleInputCtrl:=		(eInputSource:=E_IO2_InputSource.SENSOR,	sInputName:='Case Complete',
																						eTypeInput1:=E_IO2_Type.NO,		tTimeOnFilter1:=t#0ms,	tTimeOffFilter1	:=t#0ms,	(**)
											 											eTypeInput2:=E_IO2_Type.NO,		tTimeOnFilter2:=t#0ms,	tTimeOffFilter2	:=t#0ms);	(**)
	st_I_CaseDischarged					: ST_IO2_DoubleInputCtrl:=		(eInputSource:=E_IO2_InputSource.SENSOR,	sInputName:='Case Discharged',
																						eTypeInput1:=E_IO2_Type.NO,		tTimeOnFilter1:=t#0ms,	tTimeOffFilter1	:=t#0ms,	(**)
											 											eTypeInput2:=E_IO2_Type.NO,		tTimeOnFilter2:=t#0ms,	tTimeOffFilter2	:=t#0ms);	(**)
	st_I_CaseLabelValidation				: ST_IO2_DoubleInputCtrl:=		(eInputSource:=E_IO2_InputSource.SENSOR,	sInputName:='Case Label Validation',
																						eTypeInput1:=E_IO2_Type.NO,		tTimeOnFilter1:=t#0ms,	tTimeOffFilter1	:=t#0ms,	(**)
											 											eTypeInput2:=E_IO2_Type.NO,		tTimeOnFilter2:=t#0ms,	tTimeOffFilter2	:=t#0ms);	(**)
(*
	st_I_LiftComplete						: ST_IO2_DoubleInputCtrl:=		(eInputSource:=SENSOR,		eTypeInput1:=E_IO2_Type.NO,		tTimeOnFilter1:=t#0ms,	tTimeOffFilter1	:=t#0ms,	(**)
											 											eTypeInput2:=E_IO2_Type.NO,		tTimeOnFilter2:=t#0ms,	tTimeOffFilter2	:=t#0ms);	(**)
	st_I_StackComplete					: ST_IO2_DoubleInputCtrl:=		(eInputSource:=SENSOR,		eTypeInput1:=E_IO2_Type.NO,		tTimeOnFilter1:=t#0ms,	tTimeOffFilter1	:=t#0ms,	(**)
											 											eTypeInput2:=E_IO2_Type.NO,		tTimeOnFilter2:=t#0ms,	tTimeOffFilter2	:=t#0ms);	(**)
	st_I_BundleCrossPushComplete		: ST_IO2_DoubleInputCtrl:=		(eInputSource:=SENSOR,		eTypeInput1:=E_IO2_Type.NO,		tTimeOnFilter1:=t#0ms,	tTimeOffFilter1	:=t#0ms,	(**)
											 											eTypeInput2:=E_IO2_Type.NO,		tTimeOnFilter2:=t#0ms,	tTimeOffFilter2	:=t#0ms);	(**)
	st_I_BundleTranferComplete			: ST_IO2_DoubleInputCtrl:=		(eInputSource:=SENSOR,		eTypeInput1:=E_IO2_Type.NO,		tTimeOnFilter1:=t#0ms,	tTimeOffFilter1	:=t#0ms,	(**)
											 											eTypeInput2:=E_IO2_Type.NO,		tTimeOnFilter2:=t#0ms,	tTimeOffFilter2	:=t#0ms);	(**)
*)

(*******************************************************************************************************************************************************)
(********************************************************Outpurs******************************************************************************)
(*******************************************************************************************************************************************************)
(*Output Config*)
	st_Q_TPDMachineRun					: ST_IO2_OutputCtrl:=			(eTypeOutput:=E_IO2_Type.NO,		tOutputDelayed:=t#0ms,		tOutputLocked:=t#0ms,	sOutputName:='TPD Machine Run');		(* *)
	st_Q_CMLConvoyerRun				: ST_IO2_OutputCtrl:=			(eTypeOutput:=E_IO2_Type.NO,		tOutputDelayed:=t#0ms,		tOutputLocked:=t#0ms,	sOutputName:='CML Convoyer Run');		(* *)
	st_Q_EUCAPreMachineRun				: ST_IO2_OutputCtrl:=			(eTypeOutput:=E_IO2_Type.NO,		tOutputDelayed:=t#0ms,		tOutputLocked:=t#0ms,	sOutputName:='EUCA Machine Run');		(* *)
	st_Q_EUCAMachineRun				: ST_IO2_OutputCtrl:=			(eTypeOutput:=E_IO2_Type.NO,		tOutputDelayed:=t#0ms,		tOutputLocked:=t#0ms,	sOutputName:='EUCA Machine Run');		(* *)
	st_Q_CaseContentOK					: ST_IO2_OutputCtrl:=			(eTypeOutput:=E_IO2_Type.NO,		tOutputDelayed:=t#0ms,		tOutputLocked:=t#0ms,	sOutputName:='Case Content OK');		(* *)
	st_Q_CaseValidationOK				: ST_IO2_OutputCtrl:=			(eTypeOutput:=E_IO2_Type.NO,		tOutputDelayed:=t#0ms,		tOutputLocked:=t#0ms,	sOutputName:='Case Validation OK');		(* *)
	st_Q_OuterValidationOK				: ST_IO2_OutputCtrl:=			(eTypeOutput:=E_IO2_Type.NO,		tOutputDelayed:=t#0ms,		tOutputLocked:=t#0ms,	sOutputName:='Outer Validation OK');		(* *)
	st_Q_LabellerInhibit					: ST_IO2_OutputCtrl:=			(eTypeOutput:=E_IO2_Type.NO,		tOutputDelayed:=t#0ms,		tOutputLocked:=t#0ms,	sOutputName:='Labeller Inhibit');		(* *)
	st_Q_SideBeltDriveBrake				: ST_IO2_OutputCtrl:=			(eTypeOutput:=E_IO2_Type.NO,		tOutputDelayed:=t#500ms,	tOutputLocked:=t#20ms,	sOutputName:='Side Belt Drive Brake');		(* *)
	st_Q_PackSeparatorDriveBrake			: ST_IO2_OutputCtrl:=			(eTypeOutput:=E_IO2_Type.NO,		tOutputDelayed:=t#200ms,	tOutputLocked:=t#100ms,sOutputName:='Pack Separator Drive Brake');		(* *)

	st_Q_CameraLightning1				: ST_IO2_OutputCtrl:=			(eTypeOutput:=E_IO2_Type.NO,		tOutputDelayed:=t#0ms,		tOutputLocked:=t#15ms,	sOutputName:='Camera Lightning 1');		(* *)
	st_Q_CameraLightning2				: ST_IO2_OutputCtrl:=			(eTypeOutput:=E_IO2_Type.NO,		tOutputDelayed:=t#0ms,		tOutputLocked:=t#15ms,	sOutputName:='Camera Lightning 2');		(* *)
	st_Q_CameraLightning3				: ST_IO2_OutputCtrl:=			(eTypeOutput:=E_IO2_Type.NO,		tOutputDelayed:=t#0ms,		tOutputLocked:=t#15ms,	sOutputName:='Camera Lightning 3');		(* *)
	st_Q_CameraLightning4				: ST_IO2_OutputCtrl:=			(eTypeOutput:=E_IO2_Type.NO,		tOutputDelayed:=t#0ms,		tOutputLocked:=t#15ms,	sOutputName:='Camera Lightning 4');		(* *)
	st_Q_CameraLightning5				: ST_IO2_OutputCtrl:=			(eTypeOutput:=E_IO2_Type.NO,		tOutputDelayed:=t#0ms,		tOutputLocked:=t#15ms,	sOutputName:='Camera Lightning 5');		(* *)
	st_Q_CameraLightning6				: ST_IO2_OutputCtrl:=			(eTypeOutput:=E_IO2_Type.NO,		tOutputDelayed:=t#0ms,		tOutputLocked:=t#15ms,	sOutputName:='Camera Lightning 6');		(* *)
	st_Q_CameraLightning7				: ST_IO2_OutputCtrl:=			(eTypeOutput:=E_IO2_Type.NO,		tOutputDelayed:=t#0ms,		tOutputLocked:=t#15ms,	sOutputName:='Camera Lightning 7');		(* *)
	st_Q_CameraLightning8				: ST_IO2_OutputCtrl:=			(eTypeOutput:=E_IO2_Type.NO,		tOutputDelayed:=t#0ms,		tOutputLocked:=t#15ms,	sOutputName:='Camera Lightning 8');		(* *)
	st_Q_CameraLightning9				: ST_IO2_OutputCtrl:=			(eTypeOutput:=E_IO2_Type.NO,		tOutputDelayed:=t#0ms,		tOutputLocked:=t#15ms,	sOutputName:='Camera Lightning 9');		(* *)
	st_Q_CameraLightning10				: ST_IO2_OutputCtrl:=			(eTypeOutput:=E_IO2_Type.NO,		tOutputDelayed:=t#0ms,		tOutputLocked:=t#15ms,	sOutputName:='Camera Lightning 10');	(* *)
	st_Q_CameraLightning11				: ST_IO2_OutputCtrl:=			(eTypeOutput:=E_IO2_Type.NO,		tOutputDelayed:=t#0ms,		tOutputLocked:=t#15ms,	sOutputName:='Camera Lightning 11');	(* *)
	st_Q_CameraLightning12				: ST_IO2_OutputCtrl:=			(eTypeOutput:=E_IO2_Type.NO,		tOutputDelayed:=t#0ms,		tOutputLocked:=t#15ms,	sOutputName:='Camera Lightning 12');	(* *)

(*Output Config for camera triggers*)
(*
	st_Q_Camera01						: ST_IO2_OutputCtrl:=			(eTypeOutput:=E_IO2_Type.NO,		tOutputDelayed:=t#0ms,		tOutputLocked:=t#0ms);		(* *)
	st_Q_Camera02						: ST_IO2_OutputCtrl:=			(eTypeOutput:=E_IO2_Type.NO,		tOutputDelayed:=t#0ms,		tOutputLocked:=t#0ms);		(* *)
	st_Q_Camera03						: ST_IO2_OutputCtrl:=			(eTypeOutput:=E_IO2_Type.NO,		tOutputDelayed:=t#0ms,		tOutputLocked:=t#0ms);		(* *)
	st_Q_Camera04						: ST_IO2_OutputCtrl:=			(eTypeOutput:=E_IO2_Type.NO,		tOutputDelayed:=t#0ms,		tOutputLocked:=t#0ms);		(* *)
	st_Q_Camera05						: ST_IO2_OutputCtrl:=			(eTypeOutput:=E_IO2_Type.NO,		tOutputDelayed:=t#0ms,		tOutputLocked:=t#0ms);		(* *)
	st_Q_Camera06						: ST_IO2_OutputCtrl:=			(eTypeOutput:=E_IO2_Type.NO,		tOutputDelayed:=t#0ms,		tOutputLocked:=t#0ms);		(* *)
	st_Q_Camera07						: ST_IO2_OutputCtrl:=			(eTypeOutput:=E_IO2_Type.NO,		tOutputDelayed:=t#0ms,		tOutputLocked:=t#0ms);		(* *)
	st_Q_Camera08						: ST_IO2_OutputCtrl:=			(eTypeOutput:=E_IO2_Type.NO,		tOutputDelayed:=t#0ms,		tOutputLocked:=t#0ms);		(* *)
	st_Q_Camera09						: ST_IO2_OutputCtrl:=			(eTypeOutput:=E_IO2_Type.NO,		tOutputDelayed:=t#0ms,		tOutputLocked:=t#0ms);		(* *)
	st_Q_Camera10						: ST_IO2_OutputCtrl:=			(eTypeOutput:=E_IO2_Type.NO,		tOutputDelayed:=t#0ms,		tOutputLocked:=t#0ms);		(* *)
	st_Q_Camera11						: ST_IO2_OutputCtrl:=			(eTypeOutput:=E_IO2_Type.NO,		tOutputDelayed:=t#0ms,		tOutputLocked:=t#0ms);		(* *)
	st_Q_Camera12						: ST_IO2_OutputCtrl:=			(eTypeOutput:=E_IO2_Type.NO,		tOutputDelayed:=t#0ms,		tOutputLocked:=t#0ms);		(* *)
*)
END_STRUCT
END_TYPE

// ---- DUTs/METS/TCPIP Address/E_TCPIP_State.TcDUT
TYPE E_TCPIP_State :
(
	E_TCPIP_IDLE,
	E_TCPIP_CONNECT,
	E_TCPIP_SEND,
	E_TCPIP_RECEIVE,
	E_TCPIP_DISCONNECT,
	E_TCPIP_CLOSEALL,
	E_TCPIP_DONE
);
END_TYPE

// ---- GVLs/Global Variables/Aliases/T_CAC_Filename.TcDUT
TYPE T_CAC_Filename : T_MaxString;
END_TYPE

// ---- GVLs/Global Variables/Aliases/T_CASE_Barcode.TcDUT
TYPE T_CASE_Barcode : T_MaxString;
END_TYPE

// ---- GVLs/Global Variables/Aliases/T_Char.TcDUT
TYPE T_Char : STRING[1];
END_TYPE

// ---- GVLs/Global Variables/Aliases/T_CHM_Filename.TcDUT
TYPE T_CHM_Filename : T_MaxString;
END_TYPE

// ---- GVLs/Global Variables/Aliases/T_CodeBATCH.TcDUT
 TYPE T_CodeBATCH : STRING[10];
END_TYPE

// ---- GVLs/Global Variables/Aliases/T_CodeBRAND.TcDUT
 TYPE T_CodeBRAND : STRING[9];
END_TYPE

// ---- GVLs/Global Variables/Aliases/T_CodeCRYPTO.TcDUT
TYPE T_CodeCRYPTO : STRING[20];
END_TYPE

// ---- GVLs/Global Variables/Aliases/T_CodeGTIN.TcDUT
TYPE T_CodeGTIN : STRING[20];
END_TYPE

// ---- GVLs/Global Variables/Aliases/T_CodeMRP.TcDUT
TYPE T_CodeMRP : STRING[8];
END_TYPE

// ---- GVLs/Global Variables/Aliases/T_CodePIT.TcDUT
TYPE T_CodePIT : STRING[7];
END_TYPE

// ---- GVLs/Global Variables/Aliases/T_CodePO.TcDUT
TYPE T_CodePO : STRING[20];
END_TYPE

// ---- GVLs/Global Variables/Aliases/T_CodePRODUCEDATE.TcDUT
 TYPE T_CodePRODUCEDATE : STRING[14];
END_TYPE

// ---- GVLs/Global Variables/Aliases/T_CodeRSKU.TcDUT
 TYPE T_CodeRSKU : STRING[9];
END_TYPE

// ---- GVLs/Global Variables/Aliases/T_CodeURL.TcDUT
TYPE T_CodeURL : STRING[20];
END_TYPE

// ---- GVLs/Global Variables/Aliases/T_DB_LongSTRING.TcDUT
TYPE T_DB_LongSTRING : STRING(1024);
END_TYPE

// ---- GVLs/Global Variables/Aliases/T_FileExtension.TcDUT
TYPE T_FileExtension : STRING[4];
END_TYPE

// ---- GVLs/Global Variables/Aliases/T_FolderName.TcDUT
TYPE T_FolderName : STRING[25];
END_TYPE

// ---- GVLs/Global Variables/Aliases/T_FolderPath.TcDUT
TYPE T_FolderPath : STRING[100];
END_TYPE

// ---- GVLs/Global Variables/Aliases/T_FSS_RejecCode.TcDUT
TYPE T_FSS_RejecCode : STRING(40);
END_TYPE

// ---- GVLs/Global Variables/Aliases/T_HMI_PACK_Barcode.TcDUT
TYPE T_HMI_PACK_Barcode : STRING(cMAX_HMI_PACKCODE_LENGHT);
END_TYPE

// ---- GVLs/Global Variables/Aliases/T_ISO8601Time.TcDUT
TYPE T_ISO8601Time : STRING(30);
END_TYPE

// ---- GVLs/Global Variables/Aliases/T_LongSTRING.TcDUT
TYPE T_LongSTRING : STRING(1023);
END_TYPE

// ---- GVLs/Global Variables/Aliases/T_OAC_Filename.TcDUT
TYPE T_OAC_Filename : T_MaxString;
END_TYPE

// ---- GVLs/Global Variables/Aliases/T_OCV_Filename.TcDUT
TYPE T_OCV_Filename : T_MaxString;
END_TYPE

// ---- GVLs/Global Variables/Aliases/T_OHM_Filename.TcDUT
TYPE T_OHM_Filename : STRING(44);
END_TYPE

// ---- GVLs/Global Variables/Aliases/T_OUTER_Barcode.TcDUT
TYPE T_OUTER_Barcode : T_MaxString;
END_TYPE

// ---- GVLs/Global Variables/Aliases/T_PACK_Barcode.TcDUT
TYPE T_PACK_Barcode : STRING(cMAX_PACKCODE_LENGHT);
END_TYPE

// ---- GVLs/Global Variables/Aliases/T_PCM_Filename.TcDUT
 TYPE T_PCM_Filename : T_MaxString;
END_TYPE

// ---- GVLs/Global Variables/Aliases/T_PositiveDINT.TcDUT
TYPE T_PositiveDINT : DINT(0..2147483647); END_TYPE

// ---- GVLs/Global Variables/Aliases/T_PositiveINT.TcDUT
TYPE T_PositiveINT : INT(0..32767); END_TYPE

// ---- GVLs/Global Variables/Aliases/T_ProductDescription.TcDUT
TYPE T_ProductDescription : STRING[48];
END_TYPE

// ---- GVLs/Global Variables/Aliases/T_RejectCode.TcDUT
TYPE T_RejectCode : STRING[100];
END_TYPE

// ---- GVLs/Global Variables/Aliases/T_TimeLog.TcDUT
TYPE T_TimeLog : STRING[15];
END_TYPE

// ---- GVLs/Global Variables/gMessage.TcGVL
{attribute 'qualified_only'}
{attribute 'Tc2GvlVarNames'}
VAR_GLOBAL

(************************************************************************************)

	aAlarms 			: ARRAY [0..cMAX_ALARM_GROUP] OF ST_Alarms;
	aAlarmsSettings 	: ARRAY [0..cMAX_ALARM_GROUP] OF ST_AlarmSettings;

	stAlarmTable		: ST_AlarmsTable;
	stAlarmStatus		: ST_AlarmStatus;
	
(**Alarms DWord releted to Infeed Case Packer Sequence**************)

	bAlarm_PackCodeDataInvalid					: BOOL;
	bAlarm_ConsecutivePackCodeDataInvalid		: BOOL;
	bAlarm_DuplicatePackCode					: BOOL;(*bAlarm_DuplicatePackCode*)

	bWarning_DuplicatePackCode					: BOOL;
	bWarning_DuplicateOCVRemoved				: BOOL;
	bWarning_OCVStackOutOfSequence				: BOOL;
	bAlarm_ConsecutiveOCVStackOutOfSeq			: BOOL;

	bWarning_OCVArmOutOfSequence				: BOOL;
	bWarning_OCVContentRepairing				: BOOL;
	bAlarm_ConsecutiveOCVMissing				: BOOL;

	bAlarm_ConsecutiveIntermediateNoRead		: BOOL;
	bAlarm_DuplicateIntermediateCode			: BOOL;

	bWarning_TwoOutersInAggregationArea			: BOOL; (*used in SFLX*)
	bAlarm_OuterAtChuteExitNotConfirmed			: BOOL;	(*used in SFLX*)
	bAlarm_OuterRejectNotConfirmed				: BOOL;
	bAlarm_OuterDataInvalide					: BOOL;
	bAlarm_ConsecutiveOuterRejects				: BOOL;
	bAlarm_DuplicateOuterLabel					: BOOL;
	bWarning_DuplicateOACRemoved				: BOOL;

	bAlarm_InfeedQueueInvalideData				: BOOL;
	bAlarm_InfeedQueueDuplicateData				: BOOL;
	bWarning_CaseContentMissing					: BOOL;(*bWarning_CaseContentMissing*)
	bAlarm_CaseContentNotFound					: BOOL;(*bAlarm_CaseContentNotFound*)
	bAlarm_ConsecutiveCaseContentMissing		: BOOL;(*bAlarm_ConsecutiveCaseContentMissing*)
	bAlarm_DuplicateCaseContentLabel			: BOOL; (*bAlarm_DuplicateCaseLabel*)
	bAlarm_CaseContentDataInvalide				: BOOL; (*bAlarm_CaseLabelInvalidData*)
	bWarrning_DuplicatesFoundInCase				: BOOL; (*stCaseQueue.stPrintCHMData.GenericHierarchy.CaseItem.RejectReason*)

	nAlarm_DataOverWrittenInCaseQueue			: BYTE;(*nAlarm_DataOverWrittenInCaseQueue*)

	bAlarm_CaseLabelInvalidData					: BOOL;
	bAlarm_ConsecutiveCaseRejects				: BOOL;
	bAlarm_DuplicateCaseLabel					: BOOL;
	nDuplicateCaseLabelIndex					: INT;
	bWarning_CaseReanimating					: BOOL;(*bWarning_CaseReanimating*)
	bWarning_OutersTooClose						: BOOL;

	(*bAlarm_CaseRejectedData				: BOOL;*)

(* *********************************************************** *)
(* *********           Printer alarms            	 ********* *)
(* *********************************************************** *)

	bAlarm_PrinterError				: BOOL;
	bAlarm_PritnerComms				: BOOL;

(* *********************************************************** *)
(* *********      Global DB Error  alarms flag       ********* *)
(* *********************************************************** *)

	bAlarm_AuxPCVCheckDBError			: BOOL;
	bAlarm_PCVCheckDBError				: BOOL;
	bAlarm_OCVCheckDBError				: BOOL;
	bAlarm_OACCheckDBError				: BOOL;
	bAlarm_OACCaseCheckDBError			: BOOL;
	bAlarm_CACCheckDBError				: BOOL;

(* *********************************************************** *)
(* *********           G03_EtherCAT alarms           ********* *)
(* *********************************************************** *)

	bAlarm_EtherCAT_IO_Error			: BOOL;

(* *********************************************************** *)
(* *********           NV memory overlap alarms           ********* *)
(* *********************************************************** *)

	nAlarm_OverlapNVMemCheck			: WORD;
	nAlarm_OverlapBitDisplay			: WORD;

END_VAR

// ---- GVLs/Global Variables/InputsOutputs_CML/IOVariablesCX_CML.TcGVL
{attribute 'Tc2GvlVarNames'}
VAR_GLOBAL
(***************************Terminal States Diagnostic********************************)

	istEtherCATMasterState					AT	%I*	: ST_CX_EtherCATMasterState;
	iaEtherCATSlaveState					AT 	%I*	: ARRAY [0..cMAX_ETHERCAT_SLAVES] OF UINT;

(*****************************Input/Output Cards***********************************)

(*CX - Main unit*)
	(*TERMINAL 46KF2 (EK1200-5000 EtherCAT Power supply (2A E-Bus)) *****************************************)

(*TERMINAL 50KF1 (EL6001 Interface (RS232))  ********1-Channel Serial Interface RS232*****************)
	(*ib50KF1_EL6001PortNo								AT%I*: UINT;
	ist50KF1_HandScannerCOMPortDataIn					AT%I*: EL6InData22B;
	qst50KF1_HandScannerCOMPortDataOut					AT%Q*: EL6OutData22B;*)

(*TERMINAL 60KF1 - EL1008 ******************************************************)
	ib60KF1_1_AirPressureOK 							AT %I* : BOOL; (* 60KF1_1 *)
	ib60KF1_5_24VSupplyOK								AT %I* : BOOL; (* 60KF1_5 *)
	ib60KF1_2_PSRIsResetSignal							AT %I* : BOOL; (* 60KF1_2 *)
	ib60KF1_6_PSRIsOkaySignal							AT %I* : BOOL; (* 60KF1_6 *)
	ib60KF1_3_EmergancyStopSignal						AT %I* : BOOL; (* 60KF1_3 *)
	ib60KF1_7_EmergancyCircuitSignal						AT %I* : BOOL; (* 60KF1_7 *)
	ib60KF1_4_NetworkOK								AT %I* : BOOL; (* 60KF1_4 *)
	ib60KF1_8_Spare									AT %I* : BOOL; (* 60KF1_8 *)

(*TERMINAL 80KF1 - EL2008 ******************************************************)
	qb80KF1_1_SafetyResetSignal							AT %Q* : BOOL; (* 80KF1_1 *)
	qb80KF1_5_AdditionalSafetyResetSignal					AT %Q* : BOOL; (* 80KF1_5 *)
	qb80KF1_2_Spare									AT %Q* : BOOL; (* 80KF1_2 *)
	qb80KF1_6_Spare									AT %Q* : BOOL; (* 80KF1_6 *)
	qb80KF1_3_Spare									AT %Q* : BOOL; (* 80KF1_3 *)
	qb80KF1_7_Spare									AT %Q* : BOOL; (* 80KF1_7 *)
	qb80KF1_4_Spare									AT %Q* : BOOL; (* 80KF1_4 *)
	qb80KF1_8_Spare									AT %Q* : BOOL; (* 80KF1_8 *)

(*TERMINAL 95KF1 - EL6631 -  PROFINET IO Controller **************************************************)

	ist95KF1_Master01PNetState 							AT %I* : ST_CX_EtherCATMasterPNetState;

	(*DRIVE  403T1  - G120C *************************************************************************)
	ist403T1_infeedconveyor								AT %I* : ST_DRIVE_INPUT;
	qst403T1_infeedconveyor								AT %Q* : ST_DRIVE_OUTPUT;

	(*DRIVE  405T1  - G120C *************************************************************************)
	ist405T1_loweratorbelts								AT %I* : ST_DRIVE_INPUT;
	qst405T1_loweratorbelts								AT %Q* : ST_DRIVE_OUTPUT;

(*DRIVE  406T1  - G120C ******************************************************************************)
	ist406T1_rotarytransfer								AT %I* : ST_DRIVE_INPUT;
	qst406T1_rotarytransfer								AT %Q* : ST_DRIVE_OUTPUT;

(*DRIVE  407T1  - G120C ******************************************************************************)
	ist407T1_rejectconveyor								AT %I* : ST_DRIVE_INPUT;
	qst407T1_rejectconveyor								AT %Q* : ST_DRIVE_OUTPUT;

(*DRIVE  408T1  - G120C ******************************************************************************)
	ist408T1_slowdownmotors							AT %I* : ST_DRIVE_INPUT;
	qst408T1_slowdownmotors							AT %Q* : ST_DRIVE_OUTPUT;

(*DIS inputs 46KF2 (CX2100 Power Supply) ******************************************)

	ib446KF2_Up						 				AT %I* : BOOL;
	ib446KF2_Down		 							AT %I* : BOOL;
	ib446KF2_Left		 								AT %I* : BOOL;
	ib446KF2_Right	 									AT %I* : BOOL;
	ib446KF2_Enter	 									AT %I* : BOOL;

(*METS CML*)
	(*TERMINAL 446KF2 (EK1200-5000 EtherCAT Power supply (2A E-Bus)) *****************************************)

(*TERMINAL447KF1 (EL9410 E-Bus Power Supplier  (Diagnostics)) ***************2A Bus Supplay***********************)

	ib447KF1_UndervoltageUs							AT%I* : BOOL;
	ib447KF1_UndervoltageUp							AT%I* : BOOL;

(*TERMINAL 460KF1 - EL1008 ***********************************************************************)
	ib460KF1_1_Guard1UpperSideAccessDoor				AT %I* : BOOL; (* 460KF1_1 *)
	ib460KF1_5_Guard2UpperDoorLabellerSide				AT %I* : BOOL; (* 460KF1_5 *)
	ib460KF1_2_Guard3OutfeedTunnel						AT %I* : BOOL; (* 460KF1_2 *)
	ib460KF1_6_Guard4ElectricalBoxInPosition				AT %I* : BOOL; (* 460KF1_6 *)
	ib460KF1_3_Guard5RejectBinLHSide						AT %I* : BOOL; (* 460KF1_3 *)
	ib460KF1_7_Guard6RejectBinRHSide						AT %I* : BOOL; (* 460KF1_7 *)
	ib460KF1_4_Guard7HTTDoorGuard						AT %I* : BOOL; (* 460KF1_4 *)
	ib460KF1_8_Spare									AT %I* : BOOL; (* 460KF1_8 *)

(*TERMINAL 461KF1 - EL1008 ***********************************************************************)
	ib461KF1_1_Guard8Labeller1InPosition					AT %I* : BOOL; (* 461KF1_1 *)
	ib461KF1_5_Guard9Labeller2InPosition					AT %I* : BOOL; (* 461KF1_5 *)
	ib461KF1_2_Guard10FrontUpperDoor					AT %I* : BOOL; (* 461KF1_2 *)
	ib461KF1_6_Guard11GuardLowerLabellerSide				AT %I* : BOOL; (* 461KF1_6 *)
	ib461KF1_3_RejectBinGuardIsReset						AT %I* : BOOL; (* 461KF1_3 *)
	ib461KF1_7_Labeller1GuardIsReset						AT %I* : BOOL; (* 461KF1_7 *)
	ib461KF1_4_Labeller2GuardIsReset						AT %I* : BOOL; (* 461KF1_4 *)
	ib461KF1_8_Spare									AT %I* : BOOL; (* 461KF1_8 *)

(*TERMINAL 462KF1 - EL1008 ***********************************************************************)
	ib462KF1_1_Labeller1Ready							AT %I* : BOOL; (* 462KF1_1 *)
	ib462KF1_5_Labeller1SummaryWarning					AT %I* : BOOL; (* 462KF1_5 *)
	ib462KF1_2_FrontCameraTrigger						AT %I* : BOOL; (* 462KF1_2 *)
	ib462KF1_6_Labeller1DataReady						AT %I* : BOOL; (* 462KF1_6 *)
	ib462KF1_3_Labeller1HomePosition						AT %I* : BOOL; (* 462KF1_3 *)
	ib462KF1_7_Labeller1LabelPrinted						AT %I* : BOOL; (* 462KF1_7 *)
	ib462KF1_4_Labeller1Error							AT %I* : BOOL; (* 462KF1_4 *)
	ib462KF1_8_Labeller1OuterAtLabeller					AT %I* : BOOL; (* 462KF1_8 *)

(*TERMINAL 463KF1 - EL1008 ***********************************************************************)
	ib463KF1_1_Labeller2Ready							AT %I* : BOOL; (*4 63KF1_1 *)
	ib463KF1_5_Labeller2SummaryWarning					AT %I* : BOOL; (* 463KF1_5 *)
	ib463KF1_2_RearCameraTrigger							AT %I* : BOOL; (* 463KF1_2 *)
	ib463KF1_6_Labeller2DataReady						AT %I* : BOOL; (* 463KF1_6 *)
	ib463KF1_3_Lebeller2HomePosition						AT %I* : BOOL; (* 463KF1_3 *)
	ib463KF1_7_Labeller2LabelPrinted						AT %I* : BOOL; (* 463KF1_7 *)
	ib463KF1_4_Labeller2Error							AT %I* : BOOL; (* 463KF1_4 *)
	ib463KF1_8_Labeller2OuterAtLabeller					AT %I* : BOOL; (* 463KF1_8 *)

(*TERMINAL 464KF1 - EL1008 ***********************************************************************)
	ib464KF1_1_RotaryTransferPackAtStopPlate				AT %I* : BOOL; (* 464KF1_1 *)
	ib464KF1_5_RotaryTransferTorqueLimiter					AT %I* : BOOL; (* 464KF1_5 *)
	ib464KF1_2_RotaryTransferDelayStop1					AT %I* : BOOL; (* 464KF1_2 *)
	ib464KF1_6_RotaryTransferDelayStop2					AT %I* : BOOL; (* 464KF1_6 *)
	ib464KF1_3_Spare									AT %I* : BOOL; (* 464KF1_3 *)
	ib464KF1_7_Spare									AT %I* : BOOL; (* 464KF1_7 *)
	ib464KF1_4_Spare									AT %I* : BOOL; (* 464KF1_4 *)
	ib464KF1_8_Spare									AT %I* : BOOL; (* 464KF1_8 *)

(*TERMINAL 465KF1 - EL1008***********************************************************************)
	ib465KF1_1_OuterAtReject							AT %I* : BOOL; (* 465KF1_1 *)
	ib465KF1_5_CMLExitBlock								AT %I* : BOOL; (* 465KF1_5 *)
	ib465KF1_2_RejectPB								AT %I* : BOOL; (* 465KF1_2 *)
	ib465KF1_6_LoweratorGuideRHLowerInPosition			AT %I* : BOOL; (* 465KF1_6 *)
	ib465KF1_3_LoweratorGuideLHLowerInPosition			AT %I* : BOOL; (* 465KF1_3 *)
	ib465KF1_7_RejectCylinderExtended					AT %I* : BOOL; (* 465KF1_7 *)
	ib465KF1_4_RejectCylinderRetracted					AT %I* : BOOL; (* 465KF1_4 *)
	ib465KF1_8_RejectBinFull								AT %I* : BOOL; (* 465KF1_8 *)

(*TERMINAL 466KF1 - EL1008***********************************************************************)
	ib466KF1_1_AdditionalConveyor1Isolator					AT %I* : BOOL; (* 466KF1_1 *)
	ib466KF1_5_AdditionalConveyor2Isolator					AT %I* : BOOL; (* 466KF1_5 *)
	ib466KF1_2_AdditionalConveyor3Isolator					AT %I* : BOOL; (* 466KF1_2 *)
	ib466KF1_6_AdditionalConveyor4ThermalOverload			AT %I* : BOOL; (* 466KF1_6 *)
	ib466KF1_3_PreLabelCameraTrigger						AT %I* : BOOL; (* 466KF1_3 *)						(*not used on C922 and C925 *)
	ib466KF1_7_PostLabelCameraTrigger					AT %I* : BOOL; (* 466KF1_7 *)						(*not used on C922 and C925 *)
	ib466KF1_4_NCWShiftRegister							AT %I* : BOOL; (* 466KF1_4 *)						(*not used on C922 and C925 *)
	ib466KF1_8_ResetPB									AT %I* : BOOL; (* 466KF1_8 *)

(*TERMINAL 467KF1 - EL1008***********************************************************************)
	ib467KF1_1_Spare									AT %I* : BOOL; (* 467KF1_1 *)
	ib467KF1_5_OutfeedCleatedConveyorTorqueLimiter		AT %I* : BOOL; (* 467KF1_5 not used *)
	ib467KF1_2_AdditionalConveyor4OK					AT %I* : BOOL; (* 467KF1_2 sofstart is happy*)
	ib467KF1_6_Spare									AT %I* : BOOL; (* 467KF1_6 *)
	ib467KF1_3_PreMachineAutorun						AT %I* : BOOL; (* 467KF1_3 *)
	ib467KF1_7_PostMachineAutorun						AT %I* : BOOL; (* 467KF1_7 *)
	ib467KF1_4_ConveyorIndexContact						AT %I* : BOOL; (* 467KF1_4 delay stop for inffed conv for packs *)
	ib467KF1_8_OutfeedCleatedConveyorTransfer				AT %I* : BOOL; (* 467KF1_8 not used *)

(*TERMINAL 468KF1 - EL1008************************************************************************)
	ib468KF1_1_HTTMinimumLevel						AT %I* : BOOL; (* 468KF1_1 *)
	ib468KF1_5_HTTDatumSwich							AT %I* : BOOL; (* 468KF1_5 *)
	ib468KF1_2_HTTPackAtStop							AT %I* : BOOL; (* 468KF1_2 *)
	ib468KF1_6_HTTPackExitBlocked						AT %I* : BOOL; (* 468KF1_6 *)
	ib468KF1_3_HTTGuideCylinderExtended					AT %I* : BOOL; (* 468KF1_3 *)
	ib468KF1_7_PackBuildBackPreMachineCutout				AT %I* : BOOL; (* 468KF1_7 *)
	ib468KF1_4_InfeedCleatedConveyorTorqueLimiter			AT %I* : BOOL; (* 468KF1_4 *)
	ib468KF1_8_InfeedCleatedConveyorTransfer				AT %I* : BOOL; (* 468KF1_8 *)

(*TERMINAL 469KF1 - EL1008************************************************************************)
	ib469KF1_1_HTT2MinimumLevel						AT %I* : BOOL; (* 469KF1_1 *)						(*not used on C922 and C925 *)
	ib469KF1_5_HTT2DatumSwich							AT %I* : BOOL; (* 469KF1_5 *)						(*not used on C922 and C925 *)
	ib469KF1_2_HTT2PackAtStop							AT %I* : BOOL; (* 469KF1_2 *)						(*not used on C922 and C925 *)
	ib469KF1_6_HTT2ExitBlocked							AT %I* : BOOL; (* 469KF1_6 *)						(*not used on C922 and C925 *)
	ib469KF1_3_HTT2GuideCylinderExtended					AT %I* : BOOL; (* 469KF1_3 *)						(*not used on C922 and C925 *)
	ib469KF1_7_PackBuildBack2PreMachineCutout				AT %I* : BOOL; (* 469KF1_7 *)						(*not used on C922 and C925 *)
	ib469KF1_4_PreMachineHTT2ConveyorRun				AT %I* : BOOL; (* 469KF1_4 *)						(*not used on C922 and C925 *)
	ib469KF1_8_Spare									AT %I* : BOOL; (* 469KF1_8 *)						(*not used on C922 and C925 *)

(*TERMINAL 480KF1 - EL2008 ************************************************************************)
	qb480KF1_1_Spare									AT %Q* : BOOL; (* 480KF1_1 *)
	qb480KF1_5_AdditionalConveyor1Run					AT %Q* : BOOL; (* 480KF1_5 *)
	qb480KF1_2_AdditionalConveyor2Run					AT %Q* : BOOL; (* 480KF1_2 *)
	qb480KF1_6_AdditionalConveyor3Run					AT %Q* : BOOL; (* 480KF1_6 *)
	qb480KF1_3_AdditionalConveyor4Run					AT %Q* : BOOL; (* 480KF1_3 *)
	qb480KF1_7_Spare									AT %Q* : BOOL; (* 480KF1_7 *)
	qb480KF1_4_CleatedConveyrBrake						AT %Q* : BOOL; (* 480KF1_4 *)
	qb480KF1_8_PackSeparationMotorBrake					AT %Q* : BOOL; (* 480KF1_8 *)

(*TERMINAL 481KF1 - EL2008 ************************************************************************)
	qb481KF1_1_RejectCylinderExtend						AT %Q* : BOOL; (* 481KF1_1 *)	(*Solenoid*)
	qb481KF1_5_RejectCylinderRetract						AT %Q* : BOOL; (* 481KF1_5 *)	(*Solenoid*)
	qb481KF1_2_FrontHightResCameraPower					AT %Q* : BOOL; (* 481KF1_2 *)
	qb481KF1_6_ReartHightResCameraPower					AT %Q* : BOOL; (* 481KF1_6 *)
	qb481KF1_3_HTTGiudesCylinderExtend					AT %Q* : BOOL; (* 481KF1_3 *)	(*Solenoid*)
	qb481KF1_7_HTTGiudesCylinderRetract					AT %Q* : BOOL; (* 481KF1_7 *)	(*Solenoid*)
	qb481KF1_4_FrontHightResCameraTrigger				AT %Q* : BOOL; (* 481KF1_4 *)
	qb481KF1_8_ReartHightResCameraTrigger				AT %Q* : BOOL; (* 481KF1_8 *)

(*TERMINAL 482KF1 - EL2008 ************************************************************************)
	qb482KF1_1_RejectCameraPower						AT %Q*  : BOOL; (* 482KF1_1 *)	(*MasterListCameraPower*)
	qb482KF1_5_RejectCameraTrigger						AT %Q*  : BOOL; (* 482KF1_5 *)	(*MasterListCameraTrigger*)
	qb482KF1_2_PreLabelCameraPower						AT %Q*  : BOOL; (* 482KF1_2 *)						(*not used on C922 and C925 *)
	qb482KF1_6_PreLabelCameraTrigger						AT %Q*  : BOOL; (* 482KF1_6 *)						(*not used on C922 and C925 *)
	qb482KF1_3_PostLabelCameraPower					AT %Q*  : BOOL; (* 482KF1_3 *)						(*not used on C922 and C925 *)
	qb482KF1_7_PostLabelCameraTrigger					AT %Q*  : BOOL; (* 482KF1_7 *)						(*not used on C922 and C925 *)
	qb482KF1_4_Labbeller1ApplyAvailable					AT %Q*  : BOOL; (* 482KF1_4 *)
	qb482KF1_8_Labbeller2ApplyAvailable					AT %Q*  : BOOL; (* 482KF1_8 *)

(*TERMINAL 483KF1 - EL2008 ************************************************************************)
	qb483KF1_1_LightPoleGreen							AT %Q*  : BOOL; (* 483KF1_1 *)	(*MasterListCameraPower*)
	qb483KF1_5_LightPoleAmber							AT %Q*  : BOOL; (* 483KF1_5 *)	(*MasterListCameraTrigger*)
	qb483KF1_2_LightPoleRed							AT %Q*  : BOOL; (* 483KF1_2 *)
	qb483KF1_6_LightPoleAlarm							AT %Q*  : BOOL; (* 483KF1_6 *)
	qb483KF1_3_ResetPB								AT %Q*  : BOOL; (* 483KF1_3 *)
	qb483KF1_7_AdditionalPreMachineCutoutBeltInMotion		AT %Q*  : BOOL; (* 483KF1_7 *)
	qb483KF1_4_PreMachineCutoutSignalRelay				AT %Q*  : BOOL; (* 483KF1_4 *)
	qb483KF1_8_MachineRunSignalRelay					AT %Q*  : BOOL; (* 483KF1_8 *)

(*TERMINAL 490KF1 - EL2624 ************************************************************************)
	qb490KF1_1_Labeller1ResetSignal						AT %Q*  : BOOL; (*490KF1_1*)
	qb490KF1_2_Labeller2ResetSignal						AT %Q*  : BOOL; (*490KF1_2*)
	qb490KF1_3_Labeller1PrintSignal						AT %Q*  : BOOL; (*490KF1_3*)
	qb490KF1_4_Labeller2PrintSignal						AT %Q*  : BOOL; (*490KF1_4*)



END_VAR

// ---- GVLs/Global Variables/InputsOutputs_CML/IOVariablesEUCA_CML.TcGVL
{attribute 'Tc2GvlVarNames'}
VAR_GLOBAL

(*****************************Input/Output Cards***********************************)

(*METS EUCA (CML)*)
	(*TERMINAL 646KF2 (EK1200-5000 EtherCAT Power supply (2A E-Bus)) *****************************************)

	ib650KF1_EL6001PortNo								AT%I*: UINT;
	ist650KF1_HandScannerCOMPortDataIn					AT%I*: EL6InData22B;
	qst650KF1_HandScannerCOMPortDataOut				AT%Q*: EL6OutData22B;

(*TERMINAL 651KF1 - EL4002 ******************************************************)
	qn651KF1_1_LightingIntensityOuterValidCamera			AT %Q* : INT;
	qn651KF1_2_LightingIntensityOuterAggCamera			AT %Q* : INT;

(*TERMINAL 652KF1 - EL4002 ******************************************************)
	qn652KF1_1_LightingIntensityCaseContentCamera		AT %Q* : INT;
	qn652KF1_2_Spare											AT %Q* : INT;

(*TERMINAL 660KF1 (EL1008 **************************************************************)
	ib660KF1_1_IntermediatePushSensor 					AT %I*: BOOL;(* 660KF1_1 *)
	ib660KF1_5_RowCompleteSensor 						AT %I*: BOOL;(* 660KF1_1 *)
	ib660KF1_2_LayerCompleteSensor 						AT %I*: BOOL;(* 660KF1_1 *)
	ib660KF1_6_CaseCompleteSensor 						AT %I*: BOOL;(* 660KF1_1 *)
	ib660KF1_3_CaseDischargedSensor 						AT %I*: BOOL;(* 660KF1_1 *)
	ib660KF1_7_Spare  									AT %I*: BOOL;(* 660KF1_1 *)
	ib660KF1_4_CaseLabelValidationTrigSensor				AT %I*: BOOL;(* 660KF1_1 *)
	ib660KF1_8_CaseLabelValidationTrig_SFCP 				AT %I*: BOOL;(* 660KF1_1 *)

(*TERMINAL 661KF1 (EL1008  **************************************************************)
	ib661KF1_1_DoorOpenZone1 							AT %I*: BOOL;(* 661KF1_1 *)
	ib661KF1_5_DoorOpenZone2 							AT %I*: BOOL;(* 661KF1_1 *)
	ib661KF1_2_CasePackerAutoRun_SFCP					AT %I*: BOOL;(* 661KF1_1 *)
	ib661KF1_6_CaseRejectet_SFCP 						AT %I*: BOOL;(* 661KF1_1 *)
	ib661KF1_3_RowComplete_SFCP 						AT %I*: BOOL;(* 661KF1_1 *)
	ib661KF1_7_LayerComplete_SFCP 						AT %I*: BOOL;(* 661KF1_1 *)
	ib661KF1_4_CaseComplete_SFCP 						AT %I*: BOOL;(* 661KF1_1 *)
	ib661KF1_8_CaseDischarged_SFCP 						AT %I*: BOOL;(* 661KF1_1 *)

(*TERMINAL 662KF1 (EL1008 **************************************************************)
	ib662KF1_1_24VSupplyOkay 							AT %I*: BOOL;(* 662KF1_1 *)
	ib662KF1_5_24VSupplyOkayAdditionalSupplySpare 			AT %I*: BOOL;(* 662KF1_1 *)
	ib662KF1_2_Spare 									AT %I*: BOOL;(* 662KF1_1 *)
	ib662KF1_6_Spare 									AT %I*: BOOL;(* 662KF1_1 *)
	ib662KF1_3_IntermediatePush_SFCP 					AT %I*: BOOL;(* 662KF1_1 *)
	ib662KF1_7_AdditionalPreMachineAutorun 				AT %I*: BOOL;(* 662KF1_1 *)					(*not used on C922 and C925 *)
	ib662KF1_4_Spare 									AT %I*: BOOL;(* 662KF1_1 *)
	ib662KF1_8_Spare			 						AT %I*: BOOL;(* 662KF1_1 *)

(*TERMINAL 680KF1 (EL2008  **************************************************************)
	qb680KF1_1_OuterMasterListCamTrig 					AT %Q*: BOOL;(* 680KF1_1 *)					(*not used on C922 and C925 *)		(*rejectCamera instead*)
	qb680KF1_5_OuterAggregationCamTrig 					AT %Q*: BOOL;(* 680KF1_1 *)
	qb680KF1_2_CaseContentValidationCamTrig   				AT %Q*: BOOL;(* 680KF1_1 *)
	qb680KF1_6_CaseLabelValidationCamTrig 				AT %Q*: BOOL;(* 680KF1_1 *)
	qb680KF1_3_OuterMasterListCameraPower  				AT %Q*: BOOL;(* 680KF1_1 *)					(*not used on C922 and C925 *)		(*rejectCamera instead*)	(*qb482KF1_1_RejectCameraPower*)
	qb680KF1_7_OuterAggregationCamPower  				AT %Q*: BOOL;(* 680KF1_1 *)
	qb680KF1_4_CaseContentValidationCamPower  			AT %Q*: BOOL;(* 680KF1_1 *)
	qb680KF1_8_CaseLabelValidationCamPower  				AT %Q*: BOOL;(* 680KF1_1 *)

(*TERMINAL 681KF1 (EL2008  **************************************************************)
	qb681KF1_1_Cutout_STCP  							AT %Q*: BOOL;(* 681KF1_1 *)
	qb681KF1_5_CaseValidationOK_STCP  					AT %Q*: BOOL;(* 681KF1_1 *)
	qb681KF1_2_OuterValidationOK_STCP  					AT %Q*: BOOL;(* 681KF1_1 *)
	qb681KF1_6_CaseContentOK_STCP						AT %Q*: BOOL;(* 681KF1_1 *)					(*not used on C922 and C925 *)
	qb681KF1_3_HandScannerLightPoleGreen 				AT %Q*: BOOL;(* 681KF1_1 *)
	qb681KF1_7_HandScannerLightPoleRed  					AT %Q*: BOOL;(* 681KF1_1 *)
	qb681KF1_4_Spare  									AT %Q*: BOOL;(* 681KF1_1 *)
	qb681KF1_8_CMLConvoyerRun   						AT %Q*: BOOL;(* 681KF1_1 *)(*OuterRejetcSignal*)	(*not used on C922 and C925 *)

(*TERMINAL 682KF1 (EL2008  **************************************************************)
	qb682KF1_1_Spare 										AT %Q*: BOOL;(* 682KF1_1 *)
	qb682KF1_5_Spare  										AT %Q*: BOOL;(* 682KF1_1 *)
	qb682KF1_2_Spare  										AT %Q*: BOOL;(* 682KF1_1 *)
	qb682KF1_6_Spare											AT %Q*: BOOL;(* 682KF1_1 *)
	qb682KF1_3_PLCControlledOuterValidCamLightning		AT %Q*: BOOL;(* 682KF1_1 *)
	qb682KF1_7_PLCControlledOuterAggCamLightning		AT %Q*: BOOL;(* 682KF1_1 *)
	qb682KF1_4_PLCControlledCaseContentCamLightning  	AT %Q*: BOOL;(* 682KF1_1 *)
	qb682KF1_8_Spare   										AT %Q*: BOOL;(* 682KF1_1 *)

(*TERMINAL 690KF1 (EL9505 Power supply terminal 5V) ***************5V Power Supplay***********************)

	ib690KF1_PowerStatusOK								AT%I* : BOOL;
	ib690KF1_PowerOverloaded							AT%I* : BOOL;

END_VAR

// ---- GVLs/Global Variables/InputsOutputs_CML/IOVariablesPACAN_CML.TcGVL
{attribute 'Tc2GvlVarNames'}
VAR_GLOBAL
(*TERMINAL 860KF1 - EL1008 ***********************************************************************)
	ib860KF1_1_FockeSignalPackAggregationTriggerCAM1			AT %I* : BOOL; (* 860KF1_1 *)
	ib860KF1_5_FockeSignalPackAggregationTriggerCAM2			AT %I* : BOOL; (* 860KF1_5 *)
	ib860KF1_2_FockeSignalPackAggregationTriggerCAM3			AT %I* : BOOL; (* 860KF1_2 *)
	ib860KF1_6_FockeSignalAutoRun								AT %I* : BOOL; (* 860KF1_6 *)
	ib860KF1_3_FockeSignalServoIndex 							AT %I* : BOOL; (* 860KF1_3 *)
	ib860KF1_7_FockeSignalMachineIndex 							AT %I* : BOOL; (* 860KF1_7 *)
	ib860KF1_4_FockeSignalPackRejected 							AT %I* : BOOL; (* 860KF1_4 *)
	ib860KF1_8_Spare 											AT %I* : BOOL; (* 860KF1_8 *)

(*TERMINAL 861KF1 - EL1008 ***********************************************************************)
	ib861KF1_1_FockeSignalStackerIndex							AT %I* : BOOL; (* 861KF1_1 *)
	ib861KF1_5_FockeSignalStackerIndex2							AT %I* : BOOL; (* 861KF1_5 *)
	ib861KF1_2_FockeSignalFilmIndex								AT %I* : BOOL; (* 861KF1_2 *)
	ib861KF1_6_FockeSignalMasterListTrigger						AT %I* : BOOL; (* 861KF1_6 *)
	ib861KF1_3_FockeSignalTriggerBackupCAM1_3					AT %I* : BOOL; (* 861KF1_3 *)
	ib861KF1_7_FockeSignalElevatorCameraTrigger					AT %I* : BOOL; (* 861KF1_7 *)
	ib861KF1_4_FockeSignalIntermediateCameraTrigger				AT %I* : BOOL; (* 861KF1_4 *)
	ib861KF1_8_FockeSignalTriggerBackupCAM1_3					AT %I* : BOOL; (* 861KF1_8 *)

(*TERMINAL 862KF1 - EL1008 ***********************************************************************)
	ib862KF1_1_FockeSignalPushIntoTurret						AT %I* : BOOL; (* 862KF1_1 *)
	ib862KF1_5_FockeSignalBuildBack								AT %I* : BOOL; (* 862KF1_5 *)
	ib862KF1_2_FockeSignalInfeedServoRunning					AT %I* : BOOL; (* 862KF1_2 *)
	ib862KF1_6_FockeSignalOuterAccepted							AT %I* : BOOL; (* 862KF1_6 *)
	ib660KF1_3_FockeSignalMachineRunning						AT %I* : BOOL; (* 862KF1_3 *)
	ib862KF1_7_FockeSignalFilmPresent							AT %I* : BOOL; (* 862KF1_7 *)
	ib862KF1_4_FockeSignalLightControlCamera					AT %I* : BOOL; (* 862KF1_4 *)
	ib862KF1_8_FockeSignalPrinterReady							AT %I* : BOOL; (* 862KF1_8 *)

(*TERMINAL 863KF1 - EL1008 ***********************************************************************)
	ib863KF1_1_FockeSignalRefeedServo							AT %I* : BOOL; (* 863KF1_1 *)
	ib863KF1_5_Spare											AT %I* : BOOL; (* 863KF1_5 *)
	ib863KF1_2_Spare											AT %I* : BOOL; (* 863KF1_2 *)
	ib863KF1_6_Spare											AT %I* : BOOL; (* 863KF1_6 *)
	ib863KF1_3_24VDCOK											AT %I* : BOOL; (* 863KF1_3 *)
	ib863KF1_7_Spare											AT %I* : BOOL; (* 863KF1_7 *)
	ib863KF1_4_Spare											AT %I* : BOOL; (* 863KF1_4 *)
	ib863KF1_8_Spare											AT %I* : BOOL; (* 863KF1_8 *)


